LIN {X 55.448,Y -40.335,Z -83.216,A -90.000,B 90.000,C 0.000} C_DIS
LIN {X 55.688,Y -40.322,Z -83.552,A -90.000,B 90.000,C 0.000} C_DIS
LIN {X 55.796,Y -40.317,Z -83.715,A -90.000,B 90.000,C 0.000} C_DIS
LIN {X 55.903,Y -40.312,Z -83.888,A -90.000,B 90.000,C 0.000} C_DIS
LIN {X 55.980,Y -40.309,Z -84.022,A -90.000,B 90.000,C 0.000} C_DIS
LIN {X 56.380,Y -40.279,Z -84.724,A -90.000,B 90.000,C 0.000} C_DIS
LIN {X 56.567,Y -40.275,Z -85.049,A -90.000,B 90.000,C 0.000} C_DIS
LIN {X 56.659,Y -40.271,Z -85.172,A -90.000,B 90.000,C 0.000} C_DIS
LIN {X 56.815,Y -40.265,Z -85.391,A -90.000,B 90.000,C 0.000} C_DIS
LIN {X 56.970,Y -40.260,Z -85.627,A -90.000,B 90.000,C 0.000} C_DIS
LIN {X 57.075,Y -40.256,Z -85.792,A -90.000,B 90.000,C 0.000} C_DIS
LIN {X 58.077,Y -40.178,Z -87.383,A -90.000,B 90.000,C 0.000} C_DIS
LIN {X 58.154,Y -40.176,Z -87.509,A -90.000,B 90.000,C 0.000} C_DIS
LIN {X 58.234,Y -40.175,Z -87.644,A -90.000,B 90.000,C 0.000} C_DIS
LIN {X 58.357,Y -40.178,Z -87.857,A -90.000,B 90.000,C 0.000} C_DIS
LIN {X 58.489,Y -40.182,Z -88.102,A -90.000,B 90.000,C 0.000} C_DIS
LIN {X 58.598,Y -40.187,Z -88.331,A -90.000,B 90.000,C 0.000} C_DIS
LIN {X 58.752,Y -40.195,Z -88.665,A -90.000,B 90.000,C 0.000} C_DIS
LIN {X 58.752,Y -60.000,Z -88.665,A -90.000,B 90.000,C 0.000} C_DIS
LIN {X 62.631,Y -60.000,Z -64.637,A -90.000,B 90.000,C 0.000} C_DIS
LIN {X 62.631,Y -39.308,Z -64.637,A -90.000,B 90.000,C 0.000} C_DIS
LIN {X 62.803,Y -39.336,Z -65.056,A -90.000,B 90.000,C 0.000} C_DIS
LIN {X 62.966,Y -39.374,Z -65.497,A -90.000,B 90.000,C 0.000} C_DIS
LIN {X 63.006,Y -39.387,Z -65.615,A -90.000,B 90.000,C 0.000} C_DIS
LIN {X 63.056,Y -39.406,Z -65.776,A -90.000,B 90.000,C 0.000} C_DIS
LIN {X 63.115,Y -39.421,Z -65.986,A -90.000,B 90.000,C 0.000} C_DIS
LIN {X 63.170,Y -39.449,Z -66.179,A -90.000,B 90.000,C 0.000} C_DIS
LIN {X 63.215,Y -39.481,Z -66.369,A -90.000,B 90.000,C 0.000} C_DIS
LIN {X 63.277,Y -39.540,Z -66.686,A -90.000,B 90.000,C 0.000} C_DIS
LIN {X 63.366,Y -39.573,Z -66.956,A -90.000,B 90.000,C 0.000} C_DIS
LIN {X 63.448,Y -39.581,Z -67.122,A -90.000,B 90.000,C 0.000} C_DIS
LIN {X 63.626,Y -39.622,Z -67.462,A -90.000,B 90.000,C 0.000} C_DIS
LIN {X 63.736,Y -39.653,Z -67.698,A -90.000,B 90.000,C 0.000} C_DIS
LIN {X 63.814,Y -39.679,Z -67.903,A -90.000,B 90.000,C 0.000} C_DIS
LIN {X 63.888,Y -39.711,Z -68.118,A -90.000,B 90.000,C 0.000} C_DIS
LIN {X 63.960,Y -39.739,Z -68.344,A -90.000,B 90.000,C 0.000} C_DIS
LIN {X 64.010,Y -39.762,Z -68.538,A -90.000,B 90.000,C 0.000} C_DIS
LIN {X 64.032,Y -39.775,Z -68.642,A -90.000,B 90.000,C 0.000} C_DIS
LIN {X 64.060,Y -39.804,Z -68.761,A -90.000,B 90.000,C 0.000} C_DIS
LIN {X 64.106,Y -39.865,Z -68.997,A -90.000,B 90.000,C 0.000} C_DIS
LIN {X 64.202,Y -39.871,Z -69.126,A -90.000,B 90.000,C 0.000} C_DIS
LIN {X 64.331,Y -39.885,Z -69.319,A -90.000,B 90.000,C 0.000} C_DIS
LIN {X 64.452,Y -39.896,Z -69.517,A -90.000,B 90.000,C 0.000} C_DIS
LIN {X 64.575,Y -39.927,Z -69.720,A -90.000,B 90.000,C 0.000} C_DIS
LIN {X 64.644,Y -39.949,Z -69.846,A -90.000,B 90.000,C 0.000} C_DIS
LIN {X 64.711,Y -39.973,Z -69.977,A -90.000,B 90.000,C 0.000} C_DIS
LIN {X 64.741,Y -39.985,Z -70.038,A -90.000,B 90.000,C 0.000} C_DIS
LIN {X 64.793,Y -40.011,Z -70.157,A -90.000,B 90.000,C 0.000} C_DIS
LIN {X 64.862,Y -40.038,Z -70.334,A -90.000,B 90.000,C 0.000} C_DIS
LIN {X 64.948,Y -40.071,Z -70.569,A -90.000,B 90.000,C 0.000} C_DIS
LIN {X 65.029,Y -40.110,Z -70.831,A -90.000,B 90.000,C 0.000} C_DIS
LIN {X 65.095,Y -40.142,Z -71.055,A -90.000,B 90.000,C 0.000} C_DIS
LIN {X 65.138,Y -40.181,Z -71.197,A -90.000,B 90.000,C 0.000} C_DIS
LIN {X 65.489,Y -40.180,Z -71.479,A -90.000,B 90.000,C 0.000} C_DIS
LIN {X 65.574,Y -40.181,Z -71.552,A -90.000,B 90.000,C 0.000} C_DIS
LIN {X 65.793,Y -40.190,Z -71.768,A -90.000,B 90.000,C 0.000} C_DIS
LIN {X 65.900,Y -40.190,Z -71.880,A -90.000,B 90.000,C 0.000} C_DIS
LIN {X 65.920,Y -40.190,Z -71.903,A -90.000,B 90.000,C 0.000} C_DIS
LIN {X 66.214,Y -40.123,Z -72.021,A -90.000,B 90.000,C 0.000} C_DIS
LIN {X 66.578,Y -40.065,Z -72.162,A -90.000,B 90.000,C 0.000} C_DIS
LIN {X 66.676,Y -40.051,Z -72.204,A -90.000,B 90.000,C 0.000} C_DIS
LIN {X 66.897,Y -40.022,Z -72.304,A -90.000,B 90.000,C 0.000} C_DIS
LIN {X 67.010,Y -40.009,Z -72.360,A -90.000,B 90.000,C 0.000} C_DIS
LIN {X 67.972,Y -39.914,Z -72.867,A -90.000,B 90.000,C 0.000} C_DIS
LIN {X 68.175,Y -39.891,Z -72.982,A -90.000,B 90.000,C 0.000} C_DIS
LIN {X 68.701,Y -39.841,Z -73.302,A -90.000,B 90.000,C 0.000} C_DIS
LIN {X 68.861,Y -39.829,Z -73.407,A -90.000,B 90.000,C 0.000} C_DIS
LIN {X 68.964,Y -39.823,Z -73.479,A -90.000,B 90.000,C 0.000} C_DIS
LIN {X 69.180,Y -39.815,Z -73.639,A -90.000,B 90.000,C 0.000} C_DIS
LIN {X 69.326,Y -39.812,Z -73.753,A -90.000,B 90.000,C 0.000} C_DIS
LIN {X 69.405,Y -39.811,Z -73.818,A -90.000,B 90.000,C 0.000} C_DIS
LIN {X 69.492,Y -39.812,Z -73.891,A -90.000,B 90.000,C 0.000} C_DIS
LIN {X 69.916,Y -39.830,Z -74.281,A -90.000,B 90.000,C 0.000} C_DIS
LIN {X 70.119,Y -39.790,Z -74.354,A -90.000,B 90.000,C 0.000} C_DIS
LIN {X 70.283,Y -39.762,Z -74.421,A -90.000,B 90.000,C 0.000} C_DIS
LIN {X 70.508,Y -39.729,Z -74.526,A -90.000,B 90.000,C 0.000} C_DIS
LIN {X 70.711,Y -39.701,Z -74.624,A -90.000,B 90.000,C 0.000} C_DIS
LIN {X 71.011,Y -39.667,Z -74.789,A -90.000,B 90.000,C 0.000} C_DIS
LIN {X 71.174,Y -39.654,Z -74.889,A -90.000,B 90.000,C 0.000} C_DIS
LIN {X 71.373,Y -39.643,Z -75.025,A -90.000,B 90.000,C 0.000} C_DIS
LIN {X 71.608,Y -39.629,Z -75.193,A -90.000,B 90.000,C 0.000} C_DIS
LIN {X 71.729,Y -39.619,Z -75.284,A -90.000,B 90.000,C 0.000} C_DIS
LIN {X 72.076,Y -39.581,Z -75.549,A -90.000,B 90.000,C 0.000} C_DIS
LIN {X 72.224,Y -39.570,Z -75.678,A -90.000,B 90.000,C 0.000} C_DIS
LIN {X 72.416,Y -39.557,Z -75.848,A -90.000,B 90.000,C 0.000} C_DIS
LIN {X 72.547,Y -39.553,Z -75.976,A -90.000,B 90.000,C 0.000} C_DIS
LIN {X 72.645,Y -39.552,Z -76.075,A -90.000,B 90.000,C 0.000} C_DIS
LIN {X 72.773,Y -39.560,Z -76.196,A -90.000,B 90.000,C 0.000} C_DIS
LIN {X 72.854,Y -39.553,Z -76.248,A -90.000,B 90.000,C 0.000} C_DIS
LIN {X 73.182,Y -39.532,Z -76.475,A -90.000,B 90.000,C 0.000} C_DIS
LIN {X 73.340,Y -39.517,Z -76.596,A -90.000,B 90.000,C 0.000} C_DIS
LIN {X 73.415,Y -39.512,Z -76.659,A -90.000,B 90.000,C 0.000} C_DIS
LIN {X 73.579,Y -39.490,Z -76.774,A -90.000,B 90.000,C 0.000} C_DIS
LIN {X 73.871,Y -39.448,Z -76.998,A -90.000,B 90.000,C 0.000} C_DIS
LIN {X 74.097,Y -39.423,Z -77.189,A -90.000,B 90.000,C 0.000} C_DIS
LIN {X 74.181,Y -39.415,Z -77.265,A -90.000,B 90.000,C 0.000} C_DIS
LIN {X 74.301,Y -39.406,Z -77.378,A -90.000,B 90.000,C 0.000} C_DIS
LIN {X 74.531,Y -39.408,Z -77.577,A -90.000,B 90.000,C 0.000} C_DIS
LIN {X 74.759,Y -39.404,Z -77.780,A -90.000,B 90.000,C 0.000} C_DIS
LIN {X 74.822,Y -39.403,Z -77.835,A -90.000,B 90.000,C 0.000} C_DIS
LIN {X 75.001,Y -39.394,Z -77.985,A -90.000,B 90.000,C 0.000} C_DIS
LIN {X 75.071,Y -39.388,Z -78.045,A -90.000,B 90.000,C 0.000} C_DIS
LIN {X 75.136,Y -39.387,Z -78.100,A -90.000,B 90.000,C 0.000} C_DIS
LIN {X 75.196,Y -39.384,Z -78.154,A -90.000,B 90.000,C 0.000} C_DIS
LIN {X 75.547,Y -39.343,Z -78.421,A -90.000,B 90.000,C 0.000} C_DIS
LIN {X 75.912,Y -39.338,Z -78.674,A -90.000,B 90.000,C 0.000} C_DIS
LIN {X 76.049,Y -39.331,Z -78.780,A -90.000,B 90.000,C 0.000} C_DIS
LIN {X 76.147,Y -39.338,Z -78.854,A -90.000,B 90.000,C 0.000} C_DIS
LIN {X 76.292,Y -39.341,Z -78.955,A -90.000,B 90.000,C 0.000} C_DIS
LIN {X 76.399,Y -39.345,Z -79.035,A -90.000,B 90.000,C 0.000} C_DIS
LIN {X 76.474,Y -39.345,Z -79.072,A -90.000,B 90.000,C 0.000} C_DIS
LIN {X 76.612,Y -39.308,Z -79.080,A -90.000,B 90.000,C 0.000} C_DIS
LIN {X 76.612,Y -60.000,Z -79.080,A -90.000,B 90.000,C 0.000} C_DIS
LIN {X 88.646,Y -60.000,Z -102.744,A -90.000,B 90.000,C 0.000} C_DIS
LIN {X 88.646,Y -39.308,Z -102.744,A -90.000,B 90.000,C 0.000} C_DIS
LIN {X 88.487,Y -39.355,Z -102.950,A -90.000,B 90.000,C 0.000} C_DIS
LIN {X 88.363,Y -39.383,Z -103.144,A -90.000,B 90.000,C 0.000} C_DIS
LIN {X 88.211,Y -39.434,Z -103.399,A -90.000,B 90.000,C 0.000} C_DIS
LIN {X 88.135,Y -39.455,Z -103.567,A -90.000,B 90.000,C 0.000} C_DIS
LIN {X 88.144,Y -39.422,Z -103.771,A -90.000,B 90.000,C 0.000} C_DIS
LIN {X 88.186,Y -39.403,Z -104.002,A -90.000,B 90.000,C 0.000} C_DIS
LIN {X 88.227,Y -39.387,Z -104.294,A -90.000,B 90.000,C 0.000} C_DIS
LIN {X 88.233,Y -39.385,Z -104.347,A -90.000,B 90.000,C 0.000} C_DIS
LIN {X 88.314,Y -39.424,Z -105.037,A -90.000,B 90.000,C 0.000} C_DIS
LIN {X 88.419,Y -39.420,Z -105.520,A -90.000,B 90.000,C 0.000} C_DIS
LIN {X 88.449,Y -39.421,Z -105.676,A -90.000,B 90.000,C 0.000} C_DIS
LIN {X 88.476,Y -39.426,Z -105.847,A -90.000,B 90.000,C 0.000} C_DIS
LIN {X 88.504,Y -39.438,Z -106.079,A -90.000,B 90.000,C 0.000} C_DIS
LIN {X 88.535,Y -39.454,Z -106.359,A -90.000,B 90.000,C 0.000} C_DIS
LIN {X 88.548,Y -39.470,Z -106.548,A -90.000,B 90.000,C 0.000} C_DIS
LIN {X 88.551,Y -39.479,Z -106.637,A -90.000,B 90.000,C 0.000} C_DIS
LIN {X 88.548,Y -39.491,Z -106.855,A -90.000,B 90.000,C 0.000} C_DIS
LIN {X 88.543,Y -39.500,Z -106.987,A -90.000,B 90.000,C 0.000} C_DIS
LIN {X 88.531,Y -39.518,Z -107.213,A -90.000,B 90.000,C 0.000} C_DIS
LIN {X 88.570,Y -39.536,Z -108.068,A -90.000,B 90.000,C 0.000} C_DIS
LIN {X 88.572,Y -39.543,Z -108.276,A -90.000,B 90.000,C 0.000} C_DIS
LIN {X 88.570,Y -39.549,Z -108.401,A -90.000,B 90.000,C 0.000} C_DIS
LIN {X 88.562,Y -39.553,Z -108.539,A -90.000,B 90.000,C 0.000} C_DIS
LIN {X 88.541,Y -39.554,Z -108.748,A -90.000,B 90.000,C 0.000} C_DIS
LIN {X 88.482,Y -39.564,Z -109.136,A -90.000,B 90.000,C 0.000} C_DIS
LIN {X 88.466,Y -39.568,Z -109.229,A -90.000,B 90.000,C 0.000} C_DIS
LIN {X 88.427,Y -39.579,Z -109.423,A -90.000,B 90.000,C 0.000} C_DIS
LIN {X 88.395,Y -39.588,Z -109.560,A -90.000,B 90.000,C 0.000} C_DIS
LIN {X 88.352,Y -39.603,Z -109.716,A -90.000,B 90.000,C 0.000} C_DIS
LIN {X 88.195,Y -39.657,Z -110.247,A -90.000,B 90.000,C 0.000} C_DIS
LIN {X 88.083,Y -39.686,Z -110.755,A -90.000,B 90.000,C 0.000} C_DIS
LIN {X 88.036,Y -39.686,Z -110.940,A -90.000,B 90.000,C 0.000} C_DIS
LIN {X 87.935,Y -39.696,Z -111.368,A -90.000,B 90.000,C 0.000} C_DIS
LIN {X 87.898,Y -39.701,Z -111.506,A -90.000,B 90.000,C 0.000} C_DIS
LIN {X 87.857,Y -39.707,Z -111.652,A -90.000,B 90.000,C 0.000} C_DIS
LIN {X 87.827,Y -39.712,Z -111.749,A -90.000,B 90.000,C 0.000} C_DIS
LIN {X 87.739,Y -39.730,Z -112.014,A -90.000,B 90.000,C 0.000} C_DIS
LIN {X 87.648,Y -39.751,Z -112.263,A -90.000,B 90.000,C 0.000} C_DIS
LIN {X 87.392,Y -39.814,Z -112.904,A -90.000,B 90.000,C 0.000} C_DIS
LIN {X 87.199,Y -39.849,Z -113.373,A -90.000,B 90.000,C 0.000} C_DIS
LIN {X 86.963,Y -39.880,Z -114.044,A -90.000,B 90.000,C 0.000} C_DIS
LIN {X 86.838,Y -39.903,Z -114.404,A -90.000,B 90.000,C 0.000} C_DIS
LIN {X 86.484,Y -39.977,Z -115.313,A -90.000,B 90.000,C 0.000} C_DIS
LIN {X 86.191,Y -40.045,Z -116.068,A -90.000,B 90.000,C 0.000} C_DIS
LIN {X 86.080,Y -40.068,Z -116.381,A -90.000,B 90.000,C 0.000} C_DIS
LIN {X 85.781,Y -40.113,Z -117.455,A -90.000,B 90.000,C 0.000} C_DIS
LIN {X 85.664,Y -40.158,Z -117.908,A -90.000,B 90.000,C 0.000} C_DIS
LIN {X 85.654,Y -40.148,Z -119.002,A -90.000,B 90.000,C 0.000} C_DIS
LIN {X 85.738,Y -40.106,Z -119.512,A -90.000,B 90.000,C 0.000} C_DIS
LIN {X 85.882,Y -40.072,Z -120.318,A -90.000,B 90.000,C 0.000} C_DIS
LIN {X 85.916,Y -40.064,Z -120.518,A -90.000,B 90.000,C 0.000} C_DIS
LIN {X 86.185,Y -39.981,Z -121.579,A -90.000,B 90.000,C 0.000} C_DIS
LIN {X 86.320,Y -39.951,Z -122.101,A -90.000,B 90.000,C 0.000} C_DIS
LIN {X 86.350,Y -39.944,Z -122.221,A -90.000,B 90.000,C 0.000} C_DIS
LIN {X 86.375,Y -39.939,Z -122.333,A -90.000,B 90.000,C 0.000} C_DIS
LIN {X 86.420,Y -39.933,Z -122.564,A -90.000,B 90.000,C 0.000} C_DIS
LIN {X 86.439,Y -39.931,Z -122.680,A -90.000,B 90.000,C 0.000} C_DIS
LIN {X 86.466,Y -39.930,Z -122.867,A -90.000,B 90.000,C 0.000} C_DIS
LIN {X 86.538,Y -39.915,Z -123.170,A -90.000,B 90.000,C 0.000} C_DIS
LIN {X 86.605,Y -39.894,Z -123.462,A -90.000,B 90.000,C 0.000} C_DIS
LIN {X 86.698,Y -39.857,Z -123.886,A -90.000,B 90.000,C 0.000} C_DIS
LIN {X 86.776,Y -39.837,Z -124.221,A -90.000,B 90.000,C 0.000} C_DIS
LIN {X 86.837,Y -39.825,Z -124.544,A -90.000,B 90.000,C 0.000} C_DIS
LIN {X 86.851,Y -39.823,Z -124.642,A -90.000,B 90.000,C 0.000} C_DIS
LIN {X 86.911,Y -39.820,Z -125.137,A -90.000,B 90.000,C 0.000} C_DIS
LIN {X 86.942,Y -39.814,Z -125.415,A -90.000,B 90.000,C 0.000} C_DIS
LIN {X 87.002,Y -39.789,Z -125.978,A -90.000,B 90.000,C 0.000} C_DIS
LIN {X 87.037,Y -39.776,Z -126.427,A -90.000,B 90.000,C 0.000} C_DIS
LIN {X 87.043,Y -39.773,Z -126.548,A -90.000,B 90.000,C 0.000} C_DIS
LIN {X 87.059,Y -39.743,Z -127.669,A -90.000,B 90.000,C 0.000} C_DIS
LIN {X 87.070,Y -39.717,Z -128.497,A -90.000,B 90.000,C 0.000} C_DIS
LIN {X 87.067,Y -39.711,Z -128.686,A -90.000,B 90.000,C 0.000} C_DIS
LIN {X 87.033,Y -39.699,Z -129.362,A -90.000,B 90.000,C 0.000} C_DIS
LIN {X 87.016,Y -39.689,Z -129.846,A -90.000,B 90.000,C 0.000} C_DIS
LIN {X 86.985,Y -39.668,Z -130.819,A -90.000,B 90.000,C 0.000} C_DIS
LIN {X 86.968,Y -39.663,Z -131.089,A -90.000,B 90.000,C 0.000} C_DIS
LIN {X 86.930,Y -39.657,Z -131.584,A -90.000,B 90.000,C 0.000} C_DIS
LIN {X 86.917,Y -39.657,Z -131.766,A -90.000,B 90.000,C 0.000} C_DIS
LIN {X 86.865,Y -39.630,Z -133.147,A -90.000,B 90.000,C 0.000} C_DIS
LIN {X 86.850,Y -39.626,Z -133.400,A -90.000,B 90.000,C 0.000} C_DIS
LIN {X 86.798,Y -39.618,Z -134.106,A -90.000,B 90.000,C 0.000} C_DIS
LIN {X 86.786,Y -39.617,Z -134.285,A -90.000,B 90.000,C 0.000} C_DIS
LIN {X 86.751,Y -39.607,Z -135.000,A -90.000,B 90.000,C 0.000} C_DIS
LIN {X 86.727,Y -39.581,Z -136.202,A -90.000,B 90.000,C 0.000} C_DIS
LIN {X 86.713,Y -39.568,Z -136.863,A -90.000,B 90.000,C 0.000} C_DIS
LIN {X 86.705,Y -39.563,Z -137.178,A -90.000,B 90.000,C 0.000} C_DIS
LIN {X 86.656,Y -39.546,Z -138.299,A -90.000,B 90.000,C 0.000} C_DIS
LIN {X 86.648,Y -39.537,Z -138.633,A -90.000,B 90.000,C 0.000} C_DIS
LIN {X 86.609,Y -39.500,Z -140.528,A -90.000,B 90.000,C 0.000} C_DIS
LIN {X 86.528,Y -39.476,Z -142.113,A -90.000,B 90.000,C 0.000} C_DIS
LIN {X 86.512,Y -39.466,Z -142.548,A -90.000,B 90.000,C 0.000} C_DIS
LIN {X 86.459,Y -39.436,Z -144.152,A -90.000,B 90.000,C 0.000} C_DIS
LIN {X 86.446,Y -39.434,Z -144.366,A -90.000,B 90.000,C 0.000} C_DIS
LIN {X 86.309,Y -39.403,Z -146.328,A -90.000,B 90.000,C 0.000} C_DIS
LIN {X 86.274,Y -39.391,Z -146.931,A -90.000,B 90.000,C 0.000} C_DIS
LIN {X 86.210,Y -39.372,Z -148.070,A -90.000,B 90.000,C 0.000} C_DIS
LIN {X 86.178,Y -39.370,Z -148.420,A -90.000,B 90.000,C 0.000} C_DIS
LIN {X 86.058,Y -39.356,Z -149.672,A -90.000,B 90.000,C 0.000} C_DIS
LIN {X 85.954,Y -39.340,Z -150.710,A -90.000,B 90.000,C 0.000} C_DIS
LIN {X 85.844,Y -39.315,Z -151.917,A -90.000,B 90.000,C 0.000} C_DIS
LIN {X 85.811,Y -39.311,Z -152.221,A -90.000,B 90.000,C 0.000} C_DIS
LIN {X 85.781,Y -39.308,Z -152.460,A -90.000,B 90.000,C 0.000} C_DIS
LIN {X 85.781,Y -60.000,Z -152.460,A -90.000,B 90.000,C 0.000} C_DIS
LIN {X 87.625,Y -60.000,Z -117.678,A -90.000,B 90.000,C 0.000} C_DIS
LIN {X 87.625,Y -39.308,Z -117.678,A -90.000,B 90.000,C 0.000} C_DIS
LIN {X 87.494,Y -39.355,Z -118.185,A -90.000,B 90.000,C 0.000} C_DIS
LIN {X 87.487,Y -39.346,Z -118.824,A -90.000,B 90.000,C 0.000} C_DIS
LIN {X 87.560,Y -39.308,Z -119.270,A -90.000,B 90.000,C 0.000} C_DIS
LIN {X 87.560,Y -60.000,Z -119.270,A -90.000,B 90.000,C 0.000} C_DIS
LIN {X 30.587,Y -60.000,Z -77.495,A -90.000,B 90.000,C 0.000} C_DIS
LIN {X 30.587,Y -41.056,Z -77.495,A -90.000,B 90.000,C 0.000} C_DIS
LIN {X 30.404,Y -41.070,Z -77.561,A -90.000,B 90.000,C 0.000} C_DIS
LIN {X 30.295,Y -41.077,Z -77.600,A -90.000,B 90.000,C 0.000} C_DIS
LIN {X 29.998,Y -41.099,Z -77.706,A -90.000,B 90.000,C 0.000} C_DIS
LIN {X 29.486,Y -41.132,Z -77.891,A -90.000,B 90.000,C 0.000} C_DIS
LIN {X 29.537,Y -41.137,Z -77.762,A -90.000,B 90.000,C 0.000} C_DIS
LIN {X 29.558,Y -41.139,Z -77.701,A -90.000,B 90.000,C 0.000} C_DIS
LIN {X 29.594,Y -41.142,Z -77.571,A -90.000,B 90.000,C 0.000} C_DIS
LIN {X 29.625,Y -41.143,Z -77.418,A -90.000,B 90.000,C 0.000} C_DIS
LIN {X 29.640,Y -41.142,Z -77.302,A -90.000,B 90.000,C 0.000} C_DIS
LIN {X 29.650,Y -41.139,Z -77.160,A -90.000,B 90.000,C 0.000} C_DIS
LIN {X 29.651,Y -41.136,Z -77.100,A -90.000,B 90.000,C 0.000} C_DIS
LIN {X 29.649,Y -41.132,Z -77.002,A -90.000,B 90.000,C 0.000} C_DIS
LIN {X 29.639,Y -41.122,Z -76.875,A -90.000,B 90.000,C 0.000} C_DIS
LIN {X 29.626,Y -41.109,Z -76.782,A -90.000,B 90.000,C 0.000} C_DIS
LIN {X 29.598,Y -41.091,Z -76.645,A -90.000,B 90.000,C 0.000} C_DIS
LIN {X 29.529,Y -41.057,Z -76.375,A -90.000,B 90.000,C 0.000} C_DIS
LIN {X 29.515,Y -41.048,Z -76.323,A -90.000,B 90.000,C 0.000} C_DIS
LIN {X 29.477,Y -41.023,Z -76.201,A -90.000,B 90.000,C 0.000} C_DIS
LIN {X 29.425,Y -41.003,Z -76.063,A -90.000,B 90.000,C 0.000} C_DIS
LIN {X 29.393,Y -40.994,Z -75.990,A -90.000,B 90.000,C 0.000} C_DIS
LIN {X 29.532,Y -41.014,Z -76.194,A -90.000,B 90.000,C 0.000} C_DIS
LIN {X 29.643,Y -41.043,Z -76.364,A -90.000,B 90.000,C 0.000} C_DIS
LIN {X 29.810,Y -41.063,Z -76.611,A -90.000,B 90.000,C 0.000} C_DIS
LIN {X 30.025,Y -41.086,Z -76.913,A -90.000,B 90.000,C 0.000} C_DIS
LIN {X 30.053,Y -41.086,Z -76.949,A -90.000,B 90.000,C 0.000} C_DIS
LIN {X 30.138,Y -41.086,Z -77.050,A -90.000,B 90.000,C 0.000} C_DIS
LIN {X 30.340,Y -41.074,Z -77.258,A -90.000,B 90.000,C 0.000} C_DIS
LIN {X 30.433,Y -41.067,Z -77.354,A -90.000,B 90.000,C 0.000} C_DIS
LIN {X 30.499,Y -41.061,Z -77.417,A -90.000,B 90.000,C 0.000} C_DIS
LIN {X 30.587,Y -41.056,Z -77.495,A -90.000,B 90.000,C 0.000} C_DIS
LIN {X 30.587,Y -60.000,Z -77.495,A -90.000,B 90.000,C 0.000} C_DIS
LIN {X -30.129,Y -60.000,Z -90.405,A -90.000,B 90.000,C 0.000} C_DIS
LIN {X -30.129,Y -39.308,Z -90.405,A -90.000,B 90.000,C 0.000} C_DIS
LIN {X -30.060,Y -39.322,Z -90.255,A -90.000,B 90.000,C 0.000} C_DIS
LIN {X -30.026,Y -39.329,Z -90.188,A -90.000,B 90.000,C 0.000} C_DIS
LIN {X -29.675,Y -39.377,Z -89.547,A -90.000,B 90.000,C 0.000} C_DIS
LIN {X -29.319,Y -39.432,Z -88.890,A -90.000,B 90.000,C 0.000} C_DIS
LIN {X -29.145,Y -39.454,Z -88.576,A -90.000,B 90.000,C 0.000} C_DIS
LIN {X -28.986,Y -39.471,Z -88.271,A -90.000,B 90.000,C 0.000} C_DIS
LIN {X -28.868,Y -39.480,Z -88.057,A -90.000,B 90.000,C 0.000} C_DIS
LIN {X -28.612,Y -39.494,Z -87.640,A -90.000,B 90.000,C 0.000} C_DIS
LIN {X -28.327,Y -39.516,Z -87.218,A -90.000,B 90.000,C 0.000} C_DIS
LIN {X -27.589,Y -39.556,Z -86.145,A -90.000,B 90.000,C 0.000} C_DIS
LIN {X -27.389,Y -39.559,Z -85.861,A -90.000,B 90.000,C 0.000} C_DIS
LIN {X -27.210,Y -39.558,Z -85.619,A -90.000,B 90.000,C 0.000} C_DIS
LIN {X -27.072,Y -39.562,Z -85.433,A -90.000,B 90.000,C 0.000} C_DIS
LIN {X -26.958,Y -39.567,Z -85.288,A -90.000,B 90.000,C 0.000} C_DIS
LIN {X -26.797,Y -39.578,Z -85.093,A -90.000,B 90.000,C 0.000} C_DIS
LIN {X -25.931,Y -39.615,Z -84.059,A -90.000,B 90.000,C 0.000} C_DIS
LIN {X -25.793,Y -39.625,Z -83.892,A -90.000,B 90.000,C 0.000} C_DIS
LIN {X -25.587,Y -39.631,Z -83.657,A -90.000,B 90.000,C 0.000} C_DIS
LIN {X -25.130,Y -39.647,Z -83.139,A -90.000,B 90.000,C 0.000} C_DIS
LIN {X -24.889,Y -39.658,Z -82.874,A -90.000,B 90.000,C 0.000} C_DIS
LIN {X -23.786,Y -39.723,Z -81.715,A -90.000,B 90.000,C 0.000} C_DIS
LIN {X -23.601,Y -39.731,Z -81.527,A -90.000,B 90.000,C 0.000} C_DIS
LIN {X -22.538,Y -39.776,Z -80.520,A -90.000,B 90.000,C 0.000} C_DIS
LIN {X -22.410,Y -39.782,Z -80.403,A -90.000,B 90.000,C 0.000} C_DIS
LIN {X -21.978,Y -39.811,Z -80.028,A -90.000,B 90.000,C 0.000} C_DIS
LIN {X -21.823,Y -39.824,Z -79.901,A -90.000,B 90.000,C 0.000} C_DIS
LIN {X -21.508,Y -39.845,Z -79.657,A -90.000,B 90.000,C 0.000} C_DIS
LIN {X -21.087,Y -39.864,Z -79.336,A -90.000,B 90.000,C 0.000} C_DIS
LIN {X -20.813,Y -39.876,Z -79.144,A -90.000,B 90.000,C 0.000} C_DIS
LIN {X -20.037,Y -39.903,Z -78.615,A -90.000,B 90.000,C 0.000} C_DIS
LIN {X -19.819,Y -39.906,Z -78.471,A -90.000,B 90.000,C 0.000} C_DIS
LIN {X -19.686,Y -39.909,Z -78.388,A -90.000,B 90.000,C 0.000} C_DIS
LIN {X -18.777,Y -39.945,Z -77.863,A -90.000,B 90.000,C 0.000} C_DIS
LIN {X -18.662,Y -39.950,Z -77.800,A -90.000,B 90.000,C 0.000} C_DIS
LIN {X -18.375,Y -39.959,Z -77.650,A -90.000,B 90.000,C 0.000} C_DIS
LIN {X -17.935,Y -39.967,Z -77.446,A -90.000,B 90.000,C 0.000} C_DIS
LIN {X -17.734,Y -39.970,Z -77.354,A -90.000,B 90.000,C 0.000} C_DIS
LIN {X -17.278,Y -39.959,Z -77.155,A -90.000,B 90.000,C 0.000} C_DIS
LIN {X -17.056,Y -39.958,Z -77.069,A -90.000,B 90.000,C 0.000} C_DIS
LIN {X -16.621,Y -39.961,Z -76.915,A -90.000,B 90.000,C 0.000} C_DIS
LIN {X -16.143,Y -39.952,Z -76.752,A -90.000,B 90.000,C 0.000} C_DIS
LIN {X -15.801,Y -39.950,Z -76.647,A -90.000,B 90.000,C 0.000} C_DIS
LIN {X -15.391,Y -39.949,Z -76.525,A -90.000,B 90.000,C 0.000} C_DIS
LIN {X -14.632,Y -39.931,Z -76.306,A -90.000,B 90.000,C 0.000} C_DIS
LIN {X -14.379,Y -39.922,Z -76.244,A -90.000,B 90.000,C 0.000} C_DIS
LIN {X -14.275,Y -39.920,Z -76.221,A -90.000,B 90.000,C 0.000} C_DIS
LIN {X -13.551,Y -39.908,Z -76.081,A -90.000,B 90.000,C 0.000} C_DIS
LIN {X -12.950,Y -39.892,Z -75.968,A -90.000,B 90.000,C 0.000} C_DIS
LIN {X -12.788,Y -39.890,Z -75.943,A -90.000,B 90.000,C 0.000} C_DIS
LIN {X -12.426,Y -39.882,Z -75.904,A -90.000,B 90.000,C 0.000} C_DIS
LIN {X -12.084,Y -39.870,Z -75.874,A -90.000,B 90.000,C 0.000} C_DIS
LIN {X -11.917,Y -39.862,Z -75.860,A -90.000,B 90.000,C 0.000} C_DIS
LIN {X -11.431,Y -39.830,Z -75.824,A -90.000,B 90.000,C 0.000} C_DIS
LIN {X -11.236,Y -39.819,Z -75.814,A -90.000,B 90.000,C 0.000} C_DIS
LIN {X -10.430,Y -39.787,Z -75.797,A -90.000,B 90.000,C 0.000} C_DIS
LIN {X -9.953,Y -39.776,Z -75.803,A -90.000,B 90.000,C 0.000} C_DIS
LIN {X -8.395,Y -39.730,Z -75.831,A -90.000,B 90.000,C 0.000} C_DIS
LIN {X -8.291,Y -39.728,Z -75.835,A -90.000,B 90.000,C 0.000} C_DIS
LIN {X -7.791,Y -39.723,Z -75.867,A -90.000,B 90.000,C 0.000} C_DIS
LIN {X -6.721,Y -39.690,Z -75.945,A -90.000,B 90.000,C 0.000} C_DIS
LIN {X -5.934,Y -39.664,Z -76.004,A -90.000,B 90.000,C 0.000} C_DIS
LIN {X -5.156,Y -39.625,Z -76.074,A -90.000,B 90.000,C 0.000} C_DIS
LIN {X -5.105,Y -39.623,Z -76.080,A -90.000,B 90.000,C 0.000} C_DIS
LIN {X -4.883,Y -39.616,Z -76.109,A -90.000,B 90.000,C 0.000} C_DIS
LIN {X -4.446,Y -39.605,Z -76.169,A -90.000,B 90.000,C 0.000} C_DIS
LIN {X -3.413,Y -39.590,Z -76.324,A -90.000,B 90.000,C 0.000} C_DIS
LIN {X -2.938,Y -39.575,Z -76.399,A -90.000,B 90.000,C 0.000} C_DIS
LIN {X -1.406,Y -39.549,Z -76.683,A -90.000,B 90.000,C 0.000} C_DIS
LIN {X -0.800,Y -39.544,Z -76.800,A -90.000,B 90.000,C 0.000} C_DIS
LIN {X 1.141,Y -39.538,Z -77.195,A -90.000,B 90.000,C 0.000} C_DIS
LIN {X 1.724,Y -39.530,Z -77.317,A -90.000,B 90.000,C 0.000} C_DIS
LIN {X 4.226,Y -39.506,Z -77.870,A -90.000,B 90.000,C 0.000} C_DIS
LIN {X 4.732,Y -39.506,Z -77.980,A -90.000,B 90.000,C 0.000} C_DIS
LIN {X 5.634,Y -39.510,Z -78.189,A -90.000,B 90.000,C 0.000} C_DIS
LIN {X 7.423,Y -39.500,Z -78.615,A -90.000,B 90.000,C 0.000} C_DIS
LIN {X 8.961,Y -39.505,Z -78.996,A -90.000,B 90.000,C 0.000} C_DIS
LIN {X 9.315,Y -39.511,Z -79.081,A -90.000,B 90.000,C 0.000} C_DIS
LIN {X 9.694,Y -39.520,Z -79.171,A -90.000,B 90.000,C 0.000} C_DIS
LIN {X 10.706,Y -39.530,Z -79.420,A -90.000,B 90.000,C 0.000} C_DIS
LIN {X 11.555,Y -39.547,Z -79.647,A -90.000,B 90.000,C 0.000} C_DIS
LIN {X 11.681,Y -39.548,Z -79.676,A -90.000,B 90.000,C 0.000} C_DIS
LIN {X 12.289,Y -39.555,Z -79.818,A -90.000,B 90.000,C 0.000} C_DIS
LIN {X 13.473,Y -39.635,Z -80.066,A -90.000,B 90.000,C 0.000} C_DIS
LIN {X 14.312,Y -39.692,Z -80.269,A -90.000,B 90.000,C 0.000} C_DIS
LIN {X 14.404,Y -39.698,Z -80.291,A -90.000,B 90.000,C 0.000} C_DIS
LIN {X 14.505,Y -39.704,Z -80.310,A -90.000,B 90.000,C 0.000} C_DIS
LIN {X 15.313,Y -39.783,Z -80.450,A -90.000,B 90.000,C 0.000} C_DIS
LIN {X 16.728,Y -39.925,Z -80.711,A -90.000,B 90.000,C 0.000} C_DIS
LIN {X 16.974,Y -39.951,Z -80.757,A -90.000,B 90.000,C 0.000} C_DIS
LIN {X 17.313,Y -39.984,Z -80.798,A -90.000,B 90.000,C 0.000} C_DIS
LIN {X 17.686,Y -40.026,Z -80.839,A -90.000,B 90.000,C 0.000} C_DIS
LIN {X 18.252,Y -40.088,Z -80.889,A -90.000,B 90.000,C 0.000} C_DIS
LIN {X 19.206,Y -40.187,Z -80.968,A -90.000,B 90.000,C 0.000} C_DIS
LIN {X 19.435,Y -40.210,Z -80.983,A -90.000,B 90.000,C 0.000} C_DIS
LIN {X 20.104,Y -40.288,Z -80.976,A -90.000,B 90.000,C 0.000} C_DIS
LIN {X 20.547,Y -40.337,Z -80.971,A -90.000,B 90.000,C 0.000} C_DIS
LIN {X 20.786,Y -40.361,Z -80.951,A -90.000,B 90.000,C 0.000} C_DIS
LIN {X 21.160,Y -40.394,Z -80.908,A -90.000,B 90.000,C 0.000} C_DIS
LIN {X 21.542,Y -40.422,Z -80.836,A -90.000,B 90.000,C 0.000} C_DIS
LIN {X 21.735,Y -40.426,Z -80.736,A -90.000,B 90.000,C 0.000} C_DIS
LIN {X 21.816,Y -40.423,Z -80.670,A -90.000,B 90.000,C 0.000} C_DIS
LIN {X 22.233,Y -40.410,Z -80.331,A -90.000,B 90.000,C 0.000} C_DIS
LIN {X 21.604,Y -40.287,Z -79.959,A -90.000,B 90.000,C 0.000} C_DIS
LIN {X 21.322,Y -40.232,Z -79.789,A -90.000,B 90.000,C 0.000} C_DIS
LIN {X 21.185,Y -40.204,Z -79.700,A -90.000,B 90.000,C 0.000} C_DIS
LIN {X 21.094,Y -40.185,Z -79.637,A -90.000,B 90.000,C 0.000} C_DIS
LIN {X 20.932,Y -40.149,Z -79.515,A -90.000,B 90.000,C 0.000} C_DIS
LIN {X 20.734,Y -40.103,Z -79.351,A -90.000,B 90.000,C 0.000} C_DIS
LIN {X 20.605,Y -40.070,Z -79.234,A -90.000,B 90.000,C 0.000} C_DIS
LIN {X 20.559,Y -40.058,Z -79.191,A -90.000,B 90.000,C 0.000} C_DIS
LIN {X 20.446,Y -40.026,Z -79.075,A -90.000,B 90.000,C 0.000} C_DIS
LIN {X 20.326,Y -39.994,Z -78.943,A -90.000,B 90.000,C 0.000} C_DIS
LIN {X 20.264,Y -39.977,Z -78.871,A -90.000,B 90.000,C 0.000} C_DIS
LIN {X 20.155,Y -39.944,Z -78.736,A -90.000,B 90.000,C 0.000} C_DIS
LIN {X 20.115,Y -39.928,Z -78.683,A -90.000,B 90.000,C 0.000} C_DIS
LIN {X 20.049,Y -39.898,Z -78.583,A -90.000,B 90.000,C 0.000} C_DIS
LIN {X 19.932,Y -39.841,Z -78.389,A -90.000,B 90.000,C 0.000} C_DIS
LIN {X 19.875,Y -39.811,Z -78.286,A -90.000,B 90.000,C 0.000} C_DIS
LIN {X 19.773,Y -39.748,Z -78.073,A -90.000,B 90.000,C 0.000} C_DIS
LIN {X 19.692,Y -39.693,Z -77.888,A -90.000,B 90.000,C 0.000} C_DIS
LIN {X 19.604,Y -39.628,Z -77.672,A -90.000,B 90.000,C 0.000} C_DIS
LIN {X 19.592,Y -39.618,Z -77.639,A -90.000,B 90.000,C 0.000} C_DIS
LIN {X 19.463,Y -39.654,Z -77.448,A -90.000,B 90.000,C 0.000} C_DIS
LIN {X 19.393,Y -39.679,Z -77.329,A -90.000,B 90.000,C 0.000} C_DIS
LIN {X 19.239,Y -39.744,Z -77.052,A -90.000,B 90.000,C 0.000} C_DIS
LIN {X 19.139,Y -39.802,Z -76.844,A -90.000,B 90.000,C 0.000} C_DIS
LIN {X 19.077,Y -39.841,Z -76.706,A -90.000,B 90.000,C 0.000} C_DIS
LIN {X 19.044,Y -39.860,Z -76.626,A -90.000,B 90.000,C 0.000} C_DIS
LIN {X 18.972,Y -39.907,Z -76.438,A -90.000,B 90.000,C 0.000} C_DIS
LIN {X 18.911,Y -39.957,Z -76.253,A -90.000,B 90.000,C 0.000} C_DIS
LIN {X 18.879,Y -39.991,Z -76.138,A -90.000,B 90.000,C 0.000} C_DIS
LIN {X 18.849,Y -40.026,Z -76.021,A -90.000,B 90.000,C 0.000} C_DIS
LIN {X 18.833,Y -40.047,Z -75.953,A -90.000,B 90.000,C 0.000} C_DIS
LIN {X 18.806,Y -40.088,Z -75.812,A -90.000,B 90.000,C 0.000} C_DIS
LIN {X 18.764,Y -40.172,Z -75.548,A -90.000,B 90.000,C 0.000} C_DIS
LIN {X 18.743,Y -40.224,Z -75.384,A -90.000,B 90.000,C 0.000} C_DIS
LIN {X 18.730,Y -40.272,Z -75.239,A -90.000,B 90.000,C 0.000} C_DIS
LIN {X 18.725,Y -40.334,Z -75.039,A -90.000,B 90.000,C 0.000} C_DIS
LIN {X 18.728,Y -40.374,Z -74.895,A -90.000,B 90.000,C 0.000} C_DIS
LIN {X 18.743,Y -40.431,Z -74.699,A -90.000,B 90.000,C 0.000} C_DIS
LIN {X 18.772,Y -40.487,Z -74.492,A -90.000,B 90.000,C 0.000} C_DIS
LIN {X 18.782,Y -40.503,Z -74.433,A -90.000,B 90.000,C 0.000} C_DIS
LIN {X 18.799,Y -40.523,Z -74.342,A -90.000,B 90.000,C 0.000} C_DIS
LIN {X 18.838,Y -40.556,Z -74.160,A -90.000,B 90.000,C 0.000} C_DIS
LIN {X 18.865,Y -40.576,Z -74.053,A -90.000,B 90.000,C 0.000} C_DIS
LIN {X 18.910,Y -40.605,Z -73.899,A -90.000,B 90.000,C 0.000} C_DIS
LIN {X 18.970,Y -40.639,Z -73.710,A -90.000,B 90.000,C 0.000} C_DIS
LIN {X 19.008,Y -40.650,Z -73.612,A -90.000,B 90.000,C 0.000} C_DIS
LIN {X 19.058,Y -40.664,Z -73.493,A -90.000,B 90.000,C 0.000} C_DIS
LIN {X 19.128,Y -40.677,Z -73.344,A -90.000,B 90.000,C 0.000} C_DIS
LIN {X 19.191,Y -40.689,Z -73.222,A -90.000,B 90.000,C 0.000} C_DIS
LIN {X 19.216,Y -40.693,Z -73.176,A -90.000,B 90.000,C 0.000} C_DIS
LIN {X 19.317,Y -40.707,Z -73.005,A -90.000,B 90.000,C 0.000} C_DIS
LIN {X 19.412,Y -40.710,Z -72.864,A -90.000,B 90.000,C 0.000} C_DIS
LIN {X 19.448,Y -40.712,Z -72.812,A -90.000,B 90.000,C 0.000} C_DIS
LIN {X 19.550,Y -40.709,Z -72.673,A -90.000,B 90.000,C 0.000} C_DIS
LIN {X 19.598,Y -40.707,Z -72.612,A -90.000,B 90.000,C 0.000} C_DIS
LIN {X 19.720,Y -40.696,Z -72.470,A -90.000,B 90.000,C 0.000} C_DIS
LIN {X 19.760,Y -40.692,Z -72.426,A -90.000,B 90.000,C 0.000} C_DIS
LIN {X 19.895,Y -40.673,Z -72.289,A -90.000,B 90.000,C 0.000} C_DIS
LIN {X 20.082,Y -40.636,Z -72.108,A -90.000,B 90.000,C 0.000} C_DIS
LIN {X 20.228,Y -40.617,Z -71.979,A -90.000,B 90.000,C 0.000} C_DIS
LIN {X 20.326,Y -40.606,Z -71.898,A -90.000,B 90.000,C 0.000} C_DIS
LIN {X 20.416,Y -40.596,Z -71.829,A -90.000,B 90.000,C 0.000} C_DIS
LIN {X 20.555,Y -40.579,Z -71.731,A -90.000,B 90.000,C 0.000} C_DIS
LIN {X 20.589,Y -40.576,Z -71.708,A -90.000,B 90.000,C 0.000} C_DIS
LIN {X 20.606,Y -40.573,Z -71.696,A -90.000,B 90.000,C 0.000} C_DIS
LIN {X 20.707,Y -40.556,Z -71.634,A -90.000,B 90.000,C 0.000} C_DIS
LIN {X 20.799,Y -40.541,Z -71.582,A -90.000,B 90.000,C 0.000} C_DIS
LIN {X 21.102,Y -40.472,Z -71.427,A -90.000,B 90.000,C 0.000} C_DIS
LIN {X 21.342,Y -40.419,Z -71.321,A -90.000,B 90.000,C 0.000} C_DIS
LIN {X 21.420,Y -40.394,Z -71.293,A -90.000,B 90.000,C 0.000} C_DIS
LIN {X 21.710,Y -40.312,Z -71.205,A -90.000,B 90.000,C 0.000} C_DIS
LIN {X 21.854,Y -40.270,Z -71.172,A -90.000,B 90.000,C 0.000} C_DIS
LIN {X 21.977,Y -40.237,Z -71.150,A -90.000,B 90.000,C 0.000} C_DIS
LIN {X 22.107,Y -40.196,Z -71.130,A -90.000,B 90.000,C 0.000} C_DIS
LIN {X 22.276,Y -40.140,Z -71.110,A -90.000,B 90.000,C 0.000} C_DIS
LIN {X 22.471,Y -40.080,Z -71.093,A -90.000,B 90.000,C 0.000} C_DIS
LIN {X 22.658,Y -40.025,Z -71.085,A -90.000,B 90.000,C 0.000} C_DIS
LIN {X 22.835,Y -39.976,Z -71.087,A -90.000,B 90.000,C 0.000} C_DIS
LIN {X 22.998,Y -39.923,Z -71.077,A -90.000,B 90.000,C 0.000} C_DIS
LIN {X 23.051,Y -39.946,Z -71.053,A -90.000,B 90.000,C 0.000} C_DIS
LIN {X 23.191,Y -39.996,Z -71.005,A -90.000,B 90.000,C 0.000} C_DIS
LIN {X 23.337,Y -40.047,Z -70.961,A -90.000,B 90.000,C 0.000} C_DIS
LIN {X 23.490,Y -40.100,Z -70.924,A -90.000,B 90.000,C 0.000} C_DIS
LIN {X 23.582,Y -40.127,Z -70.911,A -90.000,B 90.000,C 0.000} C_DIS
LIN {X 23.792,Y -40.187,Z -70.886,A -90.000,B 90.000,C 0.000} C_DIS
LIN {X 23.911,Y -40.221,Z -70.877,A -90.000,B 90.000,C 0.000} C_DIS
LIN {X 24.159,Y -40.290,Z -70.874,A -90.000,B 90.000,C 0.000} C_DIS
LIN {X 24.274,Y -40.312,Z -70.877,A -90.000,B 90.000,C 0.000} C_DIS
LIN {X 24.389,Y -40.335,Z -70.886,A -90.000,B 90.000,C 0.000} C_DIS
LIN {X 24.587,Y -40.373,Z -70.909,A -90.000,B 90.000,C 0.000} C_DIS
LIN {X 24.709,Y -40.395,Z -70.929,A -90.000,B 90.000,C 0.000} C_DIS
LIN {X 24.934,Y -40.437,Z -70.978,A -90.000,B 90.000,C 0.000} C_DIS
LIN {X 25.130,Y -40.474,Z -71.029,A -90.000,B 90.000,C 0.000} C_DIS
LIN {X 25.567,Y -40.549,Z -71.153,A -90.000,B 90.000,C 0.000} C_DIS
LIN {X 25.925,Y -40.612,Z -71.273,A -90.000,B 90.000,C 0.000} C_DIS
LIN {X 25.956,Y -40.617,Z -71.284,A -90.000,B 90.000,C 0.000} C_DIS
LIN {X 25.980,Y -40.621,Z -71.293,A -90.000,B 90.000,C 0.000} C_DIS
LIN {X 26.506,Y -40.660,Z -71.487,A -90.000,B 90.000,C 0.000} C_DIS
LIN {X 26.522,Y -40.638,Z -71.289,A -90.000,B 90.000,C 0.000} C_DIS
LIN {X 26.532,Y -40.621,Z -71.187,A -90.000,B 90.000,C 0.000} C_DIS
LIN {X 26.549,Y -40.594,Z -71.044,A -90.000,B 90.000,C 0.000} C_DIS
LIN {X 26.568,Y -40.568,Z -70.913,A -90.000,B 90.000,C 0.000} C_DIS
LIN {X 26.606,Y -40.530,Z -70.723,A -90.000,B 90.000,C 0.000} C_DIS
LIN {X 26.668,Y -40.447,Z -70.449,A -90.000,B 90.000,C 0.000} C_DIS
LIN {X 26.694,Y -40.415,Z -70.348,A -90.000,B 90.000,C 0.000} C_DIS
LIN {X 26.743,Y -40.362,Z -70.181,A -90.000,B 90.000,C 0.000} C_DIS
LIN {X 26.752,Y -40.352,Z -70.154,A -90.000,B 90.000,C 0.000} C_DIS
LIN {X 26.801,Y -40.290,Z -70.011,A -90.000,B 90.000,C 0.000} C_DIS
LIN {X 26.871,Y -40.214,Z -69.841,A -90.000,B 90.000,C 0.000} C_DIS
LIN {X 26.919,Y -40.168,Z -69.738,A -90.000,B 90.000,C 0.000} C_DIS
LIN {X 26.950,Y -40.134,Z -69.674,A -90.000,B 90.000,C 0.000} C_DIS
LIN {X 26.993,Y -40.085,Z -69.590,A -90.000,B 90.000,C 0.000} C_DIS
LIN {X 27.058,Y -40.014,Z -69.472,A -90.000,B 90.000,C 0.000} C_DIS
LIN {X 27.061,Y -39.947,Z -69.343,A -90.000,B 90.000,C 0.000} C_DIS
LIN {X 27.052,Y -39.911,Z -69.271,A -90.000,B 90.000,C 0.000} C_DIS
LIN {X 27.039,Y -39.796,Z -69.085,A -90.000,B 90.000,C 0.000} C_DIS
LIN {X 27.038,Y -39.681,Z -68.905,A -90.000,B 90.000,C 0.000} C_DIS
LIN {X 27.047,Y -39.560,Z -68.717,A -90.000,B 90.000,C 0.000} C_DIS
LIN {X 27.053,Y -39.509,Z -68.652,A -90.000,B 90.000,C 0.000} C_DIS
LIN {X 27.079,Y -39.368,Z -68.482,A -90.000,B 90.000,C 0.000} C_DIS
LIN {X 27.072,Y -39.351,Z -68.307,A -90.000,B 90.000,C 0.000} C_DIS
LIN {X 27.069,Y -39.332,Z -68.164,A -90.000,B 90.000,C 0.000} C_DIS
LIN {X 27.068,Y -39.308,Z -68.042,A -90.000,B 90.000,C 0.000} C_DIS
LIN {X 27.064,Y -39.286,Z -67.914,A -90.000,B 90.000,C 0.000} C_DIS
LIN {X 27.055,Y -39.245,Z -67.733,A -90.000,B 90.000,C 0.000} C_DIS
LIN {X 27.043,Y -39.220,Z -67.619,A -90.000,B 90.000,C 0.000} C_DIS
LIN {X 27.028,Y -39.196,Z -67.510,A -90.000,B 90.000,C 0.000} C_DIS
LIN {X 27.010,Y -39.171,Z -67.406,A -90.000,B 90.000,C 0.000} C_DIS
LIN {X 26.988,Y -39.146,Z -67.307,A -90.000,B 90.000,C 0.000} C_DIS
LIN {X 26.962,Y -39.122,Z -67.213,A -90.000,B 90.000,C 0.000} C_DIS
LIN {X 26.934,Y -39.098,Z -67.124,A -90.000,B 90.000,C 0.000} C_DIS
LIN {X 26.902,Y -39.074,Z -67.039,A -90.000,B 90.000,C 0.000} C_DIS
LIN {X 26.868,Y -39.051,Z -66.960,A -90.000,B 90.000,C 0.000} C_DIS
LIN {X 26.830,Y -39.027,Z -66.884,A -90.000,B 90.000,C 0.000} C_DIS
LIN {X 26.789,Y -39.004,Z -66.814,A -90.000,B 90.000,C 0.000} C_DIS
LIN {X 26.746,Y -38.981,Z -66.747,A -90.000,B 90.000,C 0.000} C_DIS
LIN {X 26.700,Y -38.958,Z -66.686,A -90.000,B 90.000,C 0.000} C_DIS
LIN {X 26.651,Y -38.935,Z -66.628,A -90.000,B 90.000,C 0.000} C_DIS
LIN {X 26.599,Y -38.913,Z -66.575,A -90.000,B 90.000,C 0.000} C_DIS
LIN {X 26.545,Y -38.891,Z -66.525,A -90.000,B 90.000,C 0.000} C_DIS
LIN {X 26.488,Y -38.869,Z -66.480,A -90.000,B 90.000,C 0.000} C_DIS
LIN {X 26.429,Y -38.847,Z -66.439,A -90.000,B 90.000,C 0.000} C_DIS
LIN {X 26.368,Y -38.826,Z -66.402,A -90.000,B 90.000,C 0.000} C_DIS
LIN {X 26.304,Y -38.805,Z -66.369,A -90.000,B 90.000,C 0.000} C_DIS
LIN {X 26.238,Y -38.784,Z -66.339,A -90.000,B 90.000,C 0.000} C_DIS
LIN {X 26.135,Y -38.753,Z -66.302,A -90.000,B 90.000,C 0.000} C_DIS
LIN {X 25.991,Y -38.713,Z -66.265,A -90.000,B 90.000,C 0.000} C_DIS
LIN {X 25.839,Y -38.674,Z -66.241,A -90.000,B 90.000,C 0.000} C_DIS
LIN {X 25.681,Y -38.637,Z -66.231,A -90.000,B 90.000,C 0.000} C_DIS
LIN {X 25.599,Y -38.619,Z -66.230,A -90.000,B 90.000,C 0.000} C_DIS
LIN {X 25.431,Y -38.583,Z -66.238,A -90.000,B 90.000,C 0.000} C_DIS
LIN {X 25.258,Y -38.549,Z -66.258,A -90.000,B 90.000,C 0.000} C_DIS
LIN {X 25.079,Y -38.516,Z -66.289,A -90.000,B 90.000,C 0.000} C_DIS
LIN {X 24.897,Y -38.485,Z -66.331,A -90.000,B 90.000,C 0.000} C_DIS
LIN {X 24.711,Y -38.455,Z -66.382,A -90.000,B 90.000,C 0.000} C_DIS
LIN {X 24.615,Y -38.445,Z -66.407,A -90.000,B 90.000,C 0.000} C_DIS
LIN {X 24.517,Y -38.490,Z -66.430,A -90.000,B 90.000,C 0.000} C_DIS
LIN {X 24.421,Y -38.540,Z -66.464,A -90.000,B 90.000,C 0.000} C_DIS
LIN {X 24.228,Y -38.635,Z -66.538,A -90.000,B 90.000,C 0.000} C_DIS
LIN {X 24.130,Y -38.679,Z -66.577,A -90.000,B 90.000,C 0.000} C_DIS
LIN {X 23.935,Y -38.762,Z -66.663,A -90.000,B 90.000,C 0.000} C_DIS
LIN {X 23.640,Y -38.880,Z -66.803,A -90.000,B 90.000,C 0.000} C_DIS
LIN {X 23.444,Y -38.948,Z -66.904,A -90.000,B 90.000,C 0.000} C_DIS
LIN {X 23.248,Y -39.008,Z -67.011,A -90.000,B 90.000,C 0.000} C_DIS
LIN {X 23.054,Y -39.057,Z -67.122,A -90.000,B 90.000,C 0.000} C_DIS
LIN {X 22.957,Y -39.078,Z -67.180,A -90.000,B 90.000,C 0.000} C_DIS
LIN {X 22.766,Y -39.113,Z -67.297,A -90.000,B 90.000,C 0.000} C_DIS
LIN {X 22.577,Y -39.138,Z -67.418,A -90.000,B 90.000,C 0.000} C_DIS
LIN {X 22.484,Y -39.146,Z -67.480,A -90.000,B 90.000,C 0.000} C_DIS
LIN {X 22.300,Y -39.157,Z -67.605,A -90.000,B 90.000,C 0.000} C_DIS
LIN {X 22.121,Y -39.158,Z -67.731,A -90.000,B 90.000,C 0.000} C_DIS
LIN {X 21.946,Y -39.150,Z -67.859,A -90.000,B 90.000,C 0.000} C_DIS
LIN {X 21.777,Y -39.134,Z -67.988,A -90.000,B 90.000,C 0.000} C_DIS
LIN {X 21.613,Y -39.109,Z -68.116,A -90.000,B 90.000,C 0.000} C_DIS
LIN {X 21.457,Y -39.083,Z -68.244,A -90.000,B 90.000,C 0.000} C_DIS
LIN {X 21.307,Y -39.051,Z -68.371,A -90.000,B 90.000,C 0.000} C_DIS
LIN {X 21.165,Y -39.014,Z -68.496,A -90.000,B 90.000,C 0.000} C_DIS
LIN {X 21.031,Y -38.971,Z -68.619,A -90.000,B 90.000,C 0.000} C_DIS
LIN {X 20.906,Y -38.925,Z -68.738,A -90.000,B 90.000,C 0.000} C_DIS
LIN {X 20.876,Y -38.923,Z -68.768,A -90.000,B 90.000,C 0.000} C_DIS
LIN {X 20.736,Y -39.060,Z -68.911,A -90.000,B 90.000,C 0.000} C_DIS
LIN {X 20.636,Y -39.163,Z -69.021,A -90.000,B 90.000,C 0.000} C_DIS
LIN {X 20.506,Y -39.303,Z -69.176,A -90.000,B 90.000,C 0.000} C_DIS
LIN {X 20.434,Y -39.387,Z -69.272,A -90.000,B 90.000,C 0.000} C_DIS
LIN {X 20.349,Y -39.492,Z -69.402,A -90.000,B 90.000,C 0.000} C_DIS
LIN {X 20.311,Y -39.549,Z -69.479,A -90.000,B 90.000,C 0.000} C_DIS
LIN {X 20.286,Y -39.597,Z -69.548,A -90.000,B 90.000,C 0.000} C_DIS
LIN {X 20.276,Y -39.636,Z -69.608,A -90.000,B 90.000,C 0.000} C_DIS
LIN {X 20.278,Y -39.660,Z -69.648,A -90.000,B 90.000,C 0.000} C_DIS
LIN {X 20.285,Y -39.674,Z -69.671,A -90.000,B 90.000,C 0.000} C_DIS
LIN {X 20.302,Y -39.690,Z -69.701,A -90.000,B 90.000,C 0.000} C_DIS
LIN {X 20.318,Y -39.699,Z -69.718,A -90.000,B 90.000,C 0.000} C_DIS
LIN {X 20.350,Y -39.707,Z -69.739,A -90.000,B 90.000,C 0.000} C_DIS
LIN {X 20.377,Y -39.710,Z -69.750,A -90.000,B 90.000,C 0.000} C_DIS
LIN {X 20.425,Y -39.710,Z -69.760,A -90.000,B 90.000,C 0.000} C_DIS
LIN {X 20.461,Y -39.706,Z -69.763,A -90.000,B 90.000,C 0.000} C_DIS
LIN {X 20.547,Y -39.690,Z -69.760,A -90.000,B 90.000,C 0.000} C_DIS
LIN {X 20.651,Y -39.660,Z -69.745,A -90.000,B 90.000,C 0.000} C_DIS
LIN {X 20.773,Y -39.615,Z -69.716,A -90.000,B 90.000,C 0.000} C_DIS
LIN {X 20.842,Y -39.585,Z -69.696,A -90.000,B 90.000,C 0.000} C_DIS
LIN {X 20.916,Y -39.550,Z -69.673,A -90.000,B 90.000,C 0.000} C_DIS
LIN {X 21.080,Y -39.467,Z -69.615,A -90.000,B 90.000,C 0.000} C_DIS
LIN {X 21.365,Y -39.311,Z -69.500,A -90.000,B 90.000,C 0.000} C_DIS
LIN {X 21.476,Y -39.267,Z -69.466,A -90.000,B 90.000,C 0.000} C_DIS
LIN {X 21.587,Y -39.308,Z -69.415,A -90.000,B 90.000,C 0.000} C_DIS
LIN {X 21.742,Y -39.365,Z -69.344,A -90.000,B 90.000,C 0.000} C_DIS
LIN {X 21.877,Y -39.414,Z -69.289,A -90.000,B 90.000,C 0.000} C_DIS
LIN {X 22.052,Y -39.479,Z -69.230,A -90.000,B 90.000,C 0.000} C_DIS
LIN {X 22.159,Y -39.512,Z -69.201,A -90.000,B 90.000,C 0.000} C_DIS
LIN {X 22.289,Y -39.553,Z -69.172,A -90.000,B 90.000,C 0.000} C_DIS
LIN {X 22.373,Y -39.580,Z -69.155,A -90.000,B 90.000,C 0.000} C_DIS
LIN {X 22.498,Y -39.614,Z -69.135,A -90.000,B 90.000,C 0.000} C_DIS
LIN {X 22.613,Y -39.646,Z -69.122,A -90.000,B 90.000,C 0.000} C_DIS
LIN {X 22.770,Y -39.684,Z -69.074,A -90.000,B 90.000,C 0.000} C_DIS
LIN {X 22.938,Y -39.717,Z -69.029,A -90.000,B 90.000,C 0.000} C_DIS
LIN {X 23.108,Y -39.750,Z -68.993,A -90.000,B 90.000,C 0.000} C_DIS
LIN {X 23.243,Y -39.773,Z -68.967,A -90.000,B 90.000,C 0.000} C_DIS
LIN {X 23.439,Y -39.806,Z -68.942,A -90.000,B 90.000,C 0.000} C_DIS
LIN {X 23.583,Y -39.829,Z -68.928,A -90.000,B 90.000,C 0.000} C_DIS
LIN {X 23.747,Y -39.847,Z -68.915,A -90.000,B 90.000,C 0.000} C_DIS
LIN {X 23.971,Y -39.875,Z -68.908,A -90.000,B 90.000,C 0.000} C_DIS
LIN {X 24.288,Y -39.906,Z -68.915,A -90.000,B 90.000,C 0.000} C_DIS
LIN {X 24.413,Y -39.919,Z -68.921,A -90.000,B 90.000,C 0.000} C_DIS
LIN {X 24.552,Y -39.929,Z -68.933,A -90.000,B 90.000,C 0.000} C_DIS
LIN {X 24.788,Y -39.950,Z -68.962,A -90.000,B 90.000,C 0.000} C_DIS
LIN {X 24.956,Y -39.961,Z -68.987,A -90.000,B 90.000,C 0.000} C_DIS
LIN {X 25.049,Y -39.969,Z -69.004,A -90.000,B 90.000,C 0.000} C_DIS
LIN {X 25.051,Y -39.894,Z -68.824,A -90.000,B 90.000,C 0.000} C_DIS
LIN {X 25.057,Y -39.834,Z -68.678,A -90.000,B 90.000,C 0.000} C_DIS
LIN {X 25.070,Y -39.735,Z -68.471,A -90.000,B 90.000,C 0.000} C_DIS
LIN {X 25.092,Y -39.631,Z -68.279,A -90.000,B 90.000,C 0.000} C_DIS
LIN {X 25.081,Y -39.552,Z -68.131,A -90.000,B 90.000,C 0.000} C_DIS
LIN {X 25.076,Y -39.491,Z -68.015,A -90.000,B 90.000,C 0.000} C_DIS
LIN {X 25.075,Y -39.466,Z -67.973,A -90.000,B 90.000,C 0.000} C_DIS
LIN {X 25.080,Y -39.384,Z -67.837,A -90.000,B 90.000,C 0.000} C_DIS
LIN {X 25.093,Y -39.308,Z -67.726,A -90.000,B 90.000,C 0.000} C_DIS
LIN {X 25.093,Y -60.000,Z -67.726,A -90.000,B 90.000,C 0.000} C_DIS
LIN {X 16.997,Y -60.000,Z -74.977,A -90.000,B 90.000,C 0.000} C_DIS
LIN {X 16.997,Y -39.308,Z -74.977,A -90.000,B 90.000,C 0.000} C_DIS
LIN {X 16.989,Y -39.352,Z -74.866,A -90.000,B 90.000,C 0.000} C_DIS
LIN {X 16.986,Y -39.416,Z -74.666,A -90.000,B 90.000,C 0.000} C_DIS
LIN {X 16.988,Y -39.471,Z -74.499,A -90.000,B 90.000,C 0.000} C_DIS
LIN {X 17.004,Y -39.568,Z -74.218,A -90.000,B 90.000,C 0.000} C_DIS
LIN {X 17.011,Y -39.596,Z -74.142,A -90.000,B 90.000,C 0.000} C_DIS
LIN {X 17.050,Y -39.706,Z -73.815,A -90.000,B 90.000,C 0.000} C_DIS
LIN {X 17.088,Y -39.786,Z -73.574,A -90.000,B 90.000,C 0.000} C_DIS
LIN {X 17.119,Y -39.842,Z -73.409,A -90.000,B 90.000,C 0.000} C_DIS
LIN {X 17.155,Y -39.887,Z -73.261,A -90.000,B 90.000,C 0.000} C_DIS
LIN {X 17.241,Y -39.966,Z -72.962,A -90.000,B 90.000,C 0.000} C_DIS
LIN {X 17.257,Y -39.980,Z -72.914,A -90.000,B 90.000,C 0.000} C_DIS
LIN {X 17.336,Y -40.030,Z -72.697,A -90.000,B 90.000,C 0.000} C_DIS
LIN {X 17.386,Y -40.061,Z -72.573,A -90.000,B 90.000,C 0.000} C_DIS
LIN {X 17.465,Y -40.088,Z -72.401,A -90.000,B 90.000,C 0.000} C_DIS
LIN {X 17.531,Y -40.109,Z -72.268,A -90.000,B 90.000,C 0.000} C_DIS
LIN {X 17.595,Y -40.123,Z -72.151,A -90.000,B 90.000,C 0.000} C_DIS
LIN {X 17.675,Y -40.141,Z -72.014,A -90.000,B 90.000,C 0.000} C_DIS
LIN {X 17.734,Y -40.148,Z -71.917,A -90.000,B 90.000,C 0.000} C_DIS
LIN {X 17.882,Y -40.168,Z -71.693,A -90.000,B 90.000,C 0.000} C_DIS
LIN {X 18.042,Y -40.174,Z -71.473,A -90.000,B 90.000,C 0.000} C_DIS
LIN {X 18.169,Y -40.169,Z -71.318,A -90.000,B 90.000,C 0.000} C_DIS
LIN {X 18.224,Y -40.168,Z -71.252,A -90.000,B 90.000,C 0.000} C_DIS
LIN {X 18.353,Y -40.154,Z -71.110,A -90.000,B 90.000,C 0.000} C_DIS
LIN {X 18.415,Y -40.149,Z -71.046,A -90.000,B 90.000,C 0.000} C_DIS
LIN {X 18.609,Y -40.117,Z -70.854,A -90.000,B 90.000,C 0.000} C_DIS
LIN {X 18.756,Y -40.082,Z -70.718,A -90.000,B 90.000,C 0.000} C_DIS
LIN {X 18.963,Y -40.047,Z -70.539,A -90.000,B 90.000,C 0.000} C_DIS
LIN {X 19.149,Y -40.017,Z -70.392,A -90.000,B 90.000,C 0.000} C_DIS
LIN {X 19.204,Y -40.008,Z -70.351,A -90.000,B 90.000,C 0.000} C_DIS
LIN {X 19.268,Y -39.997,Z -70.305,A -90.000,B 90.000,C 0.000} C_DIS
LIN {X 19.485,Y -39.957,Z -70.159,A -90.000,B 90.000,C 0.000} C_DIS
LIN {X 19.712,Y -39.902,Z -70.028,A -90.000,B 90.000,C 0.000} C_DIS
LIN {X 19.843,Y -39.862,Z -69.962,A -90.000,B 90.000,C 0.000} C_DIS
LIN {X 20.193,Y -39.757,Z -69.795,A -90.000,B 90.000,C 0.000} C_DIS
LIN {X 20.430,Y -39.670,Z -69.706,A -90.000,B 90.000,C 0.000} C_DIS
LIN {X 20.550,Y -39.621,Z -69.666,A -90.000,B 90.000,C 0.000} C_DIS
LIN {X 20.679,Y -39.569,Z -69.628,A -90.000,B 90.000,C 0.000} C_DIS
LIN {X 20.917,Y -39.478,Z -69.568,A -90.000,B 90.000,C 0.000} C_DIS
LIN {X 21.070,Y -39.415,Z -69.536,A -90.000,B 90.000,C 0.000} C_DIS
LIN {X 21.230,Y -39.353,Z -69.508,A -90.000,B 90.000,C 0.000} C_DIS
LIN {X 21.351,Y -39.308,Z -69.491,A -90.000,B 90.000,C 0.000} C_DIS
LIN {X 21.470,Y -39.267,Z -69.476,A -90.000,B 90.000,C 0.000} C_DIS
LIN {X 21.686,Y -39.358,Z -69.453,A -90.000,B 90.000,C 0.000} C_DIS
LIN {X 21.878,Y -39.436,Z -69.442,A -90.000,B 90.000,C 0.000} C_DIS
LIN {X 22.044,Y -39.502,Z -69.441,A -90.000,B 90.000,C 0.000} C_DIS
LIN {X 22.118,Y -39.531,Z -69.444,A -90.000,B 90.000,C 0.000} C_DIS
LIN {X 22.249,Y -39.581,Z -69.458,A -90.000,B 90.000,C 0.000} C_DIS
LIN {X 22.357,Y -39.624,Z -69.482,A -90.000,B 90.000,C 0.000} C_DIS
LIN {X 22.424,Y -39.651,Z -69.505,A -90.000,B 90.000,C 0.000} C_DIS
LIN {X 22.479,Y -39.674,Z -69.534,A -90.000,B 90.000,C 0.000} C_DIS
LIN {X 22.508,Y -39.688,Z -69.555,A -90.000,B 90.000,C 0.000} C_DIS
LIN {X 22.544,Y -39.705,Z -69.591,A -90.000,B 90.000,C 0.000} C_DIS
LIN {X 22.568,Y -39.719,Z -69.631,A -90.000,B 90.000,C 0.000} C_DIS
LIN {X 22.581,Y -39.730,Z -69.675,A -90.000,B 90.000,C 0.000} C_DIS
LIN {X 22.583,Y -39.737,Z -69.723,A -90.000,B 90.000,C 0.000} C_DIS
LIN {X 22.579,Y -39.739,Z -69.758,A -90.000,B 90.000,C 0.000} C_DIS
LIN {X 22.571,Y -39.740,Z -69.793,A -90.000,B 90.000,C 0.000} C_DIS
LIN {X 22.541,Y -39.737,Z -69.870,A -90.000,B 90.000,C 0.000} C_DIS
LIN {X 22.495,Y -39.726,Z -69.951,A -90.000,B 90.000,C 0.000} C_DIS
LIN {X 22.432,Y -39.707,Z -70.038,A -90.000,B 90.000,C 0.000} C_DIS
LIN {X 22.355,Y -39.682,Z -70.130,A -90.000,B 90.000,C 0.000} C_DIS
LIN {X 22.263,Y -39.649,Z -70.227,A -90.000,B 90.000,C 0.000} C_DIS
LIN {X 22.213,Y -39.630,Z -70.276,A -90.000,B 90.000,C 0.000} C_DIS
LIN {X 22.158,Y -39.660,Z -70.327,A -90.000,B 90.000,C 0.000} C_DIS
LIN {X 22.040,Y -39.763,Z -70.430,A -90.000,B 90.000,C 0.000} C_DIS
LIN {X 21.911,Y -39.870,Z -70.537,A -90.000,B 90.000,C 0.000} C_DIS
LIN {X 21.769,Y -39.979,Z -70.646,A -90.000,B 90.000,C 0.000} C_DIS
LIN {X 21.695,Y -40.031,Z -70.701,A -90.000,B 90.000,C 0.000} C_DIS
LIN {X 21.539,Y -40.128,Z -70.813,A -90.000,B 90.000,C 0.000} C_DIS
LIN {X 21.457,Y -40.174,Z -70.869,A -90.000,B 90.000,C 0.000} C_DIS
LIN {X 21.287,Y -40.257,Z -70.983,A -90.000,B 90.000,C 0.000} C_DIS
LIN {X 21.109,Y -40.330,Z -71.097,A -90.000,B 90.000,C 0.000} C_DIS
LIN {X 20.923,Y -40.392,Z -71.212,A -90.000,B 90.000,C 0.000} C_DIS
LIN {X 20.731,Y -40.443,Z -71.326,A -90.000,B 90.000,C 0.000} C_DIS
LIN {X 20.533,Y -40.482,Z -71.439,A -90.000,B 90.000,C 0.000} C_DIS
LIN {X 20.330,Y -40.510,Z -71.552,A -90.000,B 90.000,C 0.000} C_DIS
LIN {X 20.123,Y -40.525,Z -71.662,A -90.000,B 90.000,C 0.000} C_DIS
LIN {X 19.912,Y -40.531,Z -71.771,A -90.000,B 90.000,C 0.000} C_DIS
LIN {X 19.698,Y -40.546,Z -71.877,A -90.000,B 90.000,C 0.000} C_DIS
LIN {X 19.483,Y -40.552,Z -71.980,A -90.000,B 90.000,C 0.000} C_DIS
LIN {X 19.266,Y -40.547,Z -72.080,A -90.000,B 90.000,C 0.000} C_DIS
LIN {X 19.049,Y -40.530,Z -72.176,A -90.000,B 90.000,C 0.000} C_DIS
LIN {X 18.833,Y -40.503,Z -72.267,A -90.000,B 90.000,C 0.000} C_DIS
LIN {X 18.725,Y -40.486,Z -72.311,A -90.000,B 90.000,C 0.000} C_DIS
LIN {X 18.617,Y -40.466,Z -72.353,A -90.000,B 90.000,C 0.000} C_DIS
LIN {X 18.404,Y -40.419,Z -72.434,A -90.000,B 90.000,C 0.000} C_DIS
LIN {X 18.193,Y -40.363,Z -72.510,A -90.000,B 90.000,C 0.000} C_DIS
LIN {X 17.985,Y -40.300,Z -72.579,A -90.000,B 90.000,C 0.000} C_DIS
LIN {X 17.782,Y -40.229,Z -72.641,A -90.000,B 90.000,C 0.000} C_DIS
LIN {X 17.682,Y -40.191,Z -72.670,A -90.000,B 90.000,C 0.000} C_DIS
LIN {X 17.487,Y -40.107,Z -72.722,A -90.000,B 90.000,C 0.000} C_DIS
LIN {X 17.298,Y -40.015,Z -72.765,A -90.000,B 90.000,C 0.000} C_DIS
LIN {X 17.206,Y -39.967,Z -72.784,A -90.000,B 90.000,C 0.000} C_DIS
LIN {X 17.027,Y -39.866,Z -72.815,A -90.000,B 90.000,C 0.000} C_DIS
LIN {X 16.856,Y -39.759,Z -72.837,A -90.000,B 90.000,C 0.000} C_DIS
LIN {X 16.695,Y -39.653,Z -72.850,A -90.000,B 90.000,C 0.000} C_DIS
LIN {X 16.543,Y -39.549,Z -72.853,A -90.000,B 90.000,C 0.000} C_DIS
LIN {X 16.401,Y -39.450,Z -72.846,A -90.000,B 90.000,C 0.000} C_DIS
LIN {X 16.271,Y -39.357,Z -72.827,A -90.000,B 90.000,C 0.000} C_DIS
LIN {X 16.210,Y -39.313,Z -72.814,A -90.000,B 90.000,C 0.000} C_DIS
LIN {X 16.152,Y -39.273,Z -72.798,A -90.000,B 90.000,C 0.000} C_DIS
LIN {X 16.097,Y -39.239,Z -72.779,A -90.000,B 90.000,C 0.000} C_DIS
LIN {X 16.046,Y -39.210,Z -72.756,A -90.000,B 90.000,C 0.000} C_DIS
LIN {X 15.998,Y -39.184,Z -72.731,A -90.000,B 90.000,C 0.000} C_DIS
LIN {X 15.954,Y -39.160,Z -72.703,A -90.000,B 90.000,C 0.000} C_DIS
LIN {X 15.894,Y -39.128,Z -72.655,A -90.000,B 90.000,C 0.000} C_DIS
LIN {X 15.859,Y -39.110,Z -72.618,A -90.000,B 90.000,C 0.000} C_DIS
LIN {X 15.827,Y -39.095,Z -72.579,A -90.000,B 90.000,C 0.000} C_DIS
LIN {X 15.787,Y -39.077,Z -72.513,A -90.000,B 90.000,C 0.000} C_DIS
LIN {X 15.756,Y -39.066,Z -72.440,A -90.000,B 90.000,C 0.000} C_DIS
LIN {X 15.735,Y -39.061,Z -72.358,A -90.000,B 90.000,C 0.000} C_DIS
LIN {X 15.726,Y -39.061,Z -72.299,A -90.000,B 90.000,C 0.000} C_DIS
LIN {X 15.721,Y -39.064,Z -72.237,A -90.000,B 90.000,C 0.000} C_DIS
LIN {X 15.723,Y -39.075,Z -72.136,A -90.000,B 90.000,C 0.000} C_DIS
LIN {X 15.730,Y -39.086,Z -72.064,A -90.000,B 90.000,C 0.000} C_DIS
LIN {X 15.742,Y -39.101,Z -71.988,A -90.000,B 90.000,C 0.000} C_DIS
LIN {X 15.769,Y -39.129,Z -71.867,A -90.000,B 90.000,C 0.000} C_DIS
LIN {X 15.822,Y -39.179,Z -71.692,A -90.000,B 90.000,C 0.000} C_DIS
LIN {X 15.897,Y -39.233,Z -71.500,A -90.000,B 90.000,C 0.000} C_DIS
LIN {X 15.993,Y -39.290,Z -71.291,A -90.000,B 90.000,C 0.000} C_DIS
LIN {X 16.049,Y -39.308,Z -71.179,A -90.000,B 90.000,C 0.000} C_DIS
LIN {X 16.138,Y -39.348,Z -71.008,A -90.000,B 90.000,C 0.000} C_DIS
LIN {X 16.228,Y -39.376,Z -70.851,A -90.000,B 90.000,C 0.000} C_DIS
LIN {X 16.321,Y -39.404,Z -70.700,A -90.000,B 90.000,C 0.000} C_DIS
LIN {X 16.392,Y -39.418,Z -70.591,A -90.000,B 90.000,C 0.000} C_DIS
LIN {X 16.525,Y -39.441,Z -70.395,A -90.000,B 90.000,C 0.000} C_DIS
LIN {X 16.583,Y -39.445,Z -70.316,A -90.000,B 90.000,C 0.000} C_DIS
LIN {X 16.712,Y -39.456,Z -70.149,A -90.000,B 90.000,C 0.000} C_DIS
LIN {X 16.861,Y -39.454,Z -69.972,A -90.000,B 90.000,C 0.000} C_DIS
LIN {X 16.934,Y -39.452,Z -69.888,A -90.000,B 90.000,C 0.000} C_DIS
LIN {X 17.143,Y -39.436,Z -69.669,A -90.000,B 90.000,C 0.000} C_DIS
LIN {X 17.378,Y -39.399,Z -69.439,A -90.000,B 90.000,C 0.000} C_DIS
LIN {X 17.457,Y -39.381,Z -69.368,A -90.000,B 90.000,C 0.000} C_DIS
LIN {X 17.611,Y -39.351,Z -69.238,A -90.000,B 90.000,C 0.000} C_DIS
LIN {X 17.683,Y -39.330,Z -69.179,A -90.000,B 90.000,C 0.000} C_DIS
LIN {X 17.789,Y -39.308,Z -69.096,A -90.000,B 90.000,C 0.000} C_DIS
LIN {X 17.789,Y -60.000,Z -69.096,A -90.000,B 90.000,C 0.000} C_DIS
LIN {X 13.365,Y -60.000,Z -78.022,A -90.000,B 90.000,C 0.000} C_DIS
LIN {X 13.365,Y -39.308,Z -78.022,A -90.000,B 90.000,C 0.000} C_DIS
LIN {X 13.957,Y -39.387,Z -78.141,A -90.000,B 90.000,C 0.000} C_DIS
LIN {X 14.759,Y -39.495,Z -78.330,A -90.000,B 90.000,C 0.000} C_DIS
LIN {X 14.821,Y -39.503,Z -78.345,A -90.000,B 90.000,C 0.000} C_DIS
LIN {X 15.188,Y -39.545,Z -78.408,A -90.000,B 90.000,C 0.000} C_DIS
LIN {X 15.770,Y -39.609,Z -78.509,A -90.000,B 90.000,C 0.000} C_DIS
LIN {X 17.125,Y -39.745,Z -78.760,A -90.000,B 90.000,C 0.000} C_DIS
LIN {X 17.293,Y -39.760,Z -78.791,A -90.000,B 90.000,C 0.000} C_DIS
LIN {X 17.907,Y -39.813,Z -78.862,A -90.000,B 90.000,C 0.000} C_DIS
LIN {X 17.938,Y -39.816,Z -78.865,A -90.000,B 90.000,C 0.000} C_DIS
LIN {X 17.834,Y -39.777,Z -78.623,A -90.000,B 90.000,C 0.000} C_DIS
LIN {X 17.814,Y -39.769,Z -78.573,A -90.000,B 90.000,C 0.000} C_DIS
LIN {X 17.752,Y -39.752,Z -78.478,A -90.000,B 90.000,C 0.000} C_DIS
LIN {X 17.650,Y -39.723,Z -78.310,A -90.000,B 90.000,C 0.000} C_DIS
LIN {X 17.485,Y -39.673,Z -78.011,A -90.000,B 90.000,C 0.000} C_DIS
LIN {X 17.464,Y -39.667,Z -77.972,A -90.000,B 90.000,C 0.000} C_DIS
LIN {X 17.407,Y -39.642,Z -77.850,A -90.000,B 90.000,C 0.000} C_DIS
LIN {X 17.304,Y -39.595,Z -77.612,A -90.000,B 90.000,C 0.000} C_DIS
LIN {X 17.225,Y -39.553,Z -77.405,A -90.000,B 90.000,C 0.000} C_DIS
LIN {X 17.173,Y -39.522,Z -77.248,A -90.000,B 90.000,C 0.000} C_DIS
LIN {X 17.145,Y -39.499,Z -77.149,A -90.000,B 90.000,C 0.000} C_DIS
LIN {X 17.119,Y -39.475,Z -77.054,A -90.000,B 90.000,C 0.000} C_DIS
LIN {X 17.090,Y -39.439,Z -76.924,A -90.000,B 90.000,C 0.000} C_DIS
LIN {X 17.051,Y -39.380,Z -76.707,A -90.000,B 90.000,C 0.000} C_DIS
LIN {X 17.037,Y -39.348,Z -76.594,A -90.000,B 90.000,C 0.000} C_DIS
LIN {X 17.026,Y -39.308,Z -76.455,A -90.000,B 90.000,C 0.000} C_DIS
LIN {X 17.026,Y -60.000,Z -76.455,A -90.000,B 90.000,C 0.000} C_DIS
LIN {X -26.369,Y -60.000,Z -134.517,A -90.000,B 90.000,C 0.000} C_DIS
LIN {X -26.369,Y -39.308,Z -134.517,A -90.000,B 90.000,C 0.000} C_DIS
LIN {X -26.416,Y -39.321,Z -134.425,A -90.000,B 90.000,C 0.000} C_DIS
LIN {X -26.693,Y -39.410,Z -133.851,A -90.000,B 90.000,C 0.000} C_DIS
LIN {X -27.060,Y -39.500,Z -133.040,A -90.000,B 90.000,C 0.000} C_DIS
LIN {X -27.151,Y -39.517,Z -132.816,A -90.000,B 90.000,C 0.000} C_DIS
LIN {X -27.588,Y -39.593,Z -131.700,A -90.000,B 90.000,C 0.000} C_DIS
LIN {X -27.836,Y -39.632,Z -131.076,A -90.000,B 90.000,C 0.000} C_DIS
LIN {X -28.397,Y -39.676,Z -129.828,A -90.000,B 90.000,C 0.000} C_DIS
LIN {X -28.479,Y -39.686,Z -129.631,A -90.000,B 90.000,C 0.000} C_DIS
LIN {X -28.563,Y -39.703,Z -129.407,A -90.000,B 90.000,C 0.000} C_DIS
LIN {X -28.641,Y -39.720,Z -129.184,A -90.000,B 90.000,C 0.000} C_DIS
LIN {X -28.929,Y -39.802,Z -128.285,A -90.000,B 90.000,C 0.000} C_DIS
LIN {X -28.943,Y -39.807,Z -128.239,A -90.000,B 90.000,C 0.000} C_DIS
LIN {X -29.050,Y -39.827,Z -127.910,A -90.000,B 90.000,C 0.000} C_DIS
LIN {X -29.282,Y -39.875,Z -127.173,A -90.000,B 90.000,C 0.000} C_DIS
LIN {X -29.381,Y -39.888,Z -126.842,A -90.000,B 90.000,C 0.000} C_DIS
LIN {X -29.509,Y -39.881,Z -126.529,A -90.000,B 90.000,C 0.000} C_DIS
LIN {X -29.590,Y -39.883,Z -126.339,A -90.000,B 90.000,C 0.000} C_DIS
LIN {X -29.694,Y -39.881,Z -126.089,A -90.000,B 90.000,C 0.000} C_DIS
LIN {X -29.964,Y -39.861,Z -125.425,A -90.000,B 90.000,C 0.000} C_DIS
LIN {X -30.113,Y -39.849,Z -125.063,A -90.000,B 90.000,C 0.000} C_DIS
LIN {X -30.197,Y -39.845,Z -124.837,A -90.000,B 90.000,C 0.000} C_DIS
LIN {X -30.278,Y -39.845,Z -124.595,A -90.000,B 90.000,C 0.000} C_DIS
LIN {X -30.527,Y -39.883,Z -123.876,A -90.000,B 90.000,C 0.000} C_DIS
LIN {X -30.595,Y -39.894,Z -123.678,A -90.000,B 90.000,C 0.000} C_DIS
LIN {X -30.656,Y -39.907,Z -123.482,A -90.000,B 90.000,C 0.000} C_DIS
LIN {X -30.749,Y -39.924,Z -123.161,A -90.000,B 90.000,C 0.000} C_DIS
LIN {X -30.796,Y -39.929,Z -122.991,A -90.000,B 90.000,C 0.000} C_DIS
LIN {X -30.917,Y -39.947,Z -122.567,A -90.000,B 90.000,C 0.000} C_DIS
LIN {X -30.992,Y -39.942,Z -122.393,A -90.000,B 90.000,C 0.000} C_DIS
LIN {X -31.477,Y -39.860,Z -121.227,A -90.000,B 90.000,C 0.000} C_DIS
LIN {X -31.526,Y -39.859,Z -121.117,A -90.000,B 90.000,C 0.000} C_DIS
LIN {X -31.620,Y -39.860,Z -120.882,A -90.000,B 90.000,C 0.000} C_DIS
LIN {X -31.779,Y -39.873,Z -120.422,A -90.000,B 90.000,C 0.000} C_DIS
LIN {X -31.846,Y -39.882,Z -120.205,A -90.000,B 90.000,C 0.000} C_DIS
LIN {X -31.907,Y -39.893,Z -119.991,A -90.000,B 90.000,C 0.000} C_DIS
LIN {X -32.006,Y -39.899,Z -119.622,A -90.000,B 90.000,C 0.000} C_DIS
LIN {X -32.055,Y -39.904,Z -119.428,A -90.000,B 90.000,C 0.000} C_DIS
LIN {X -32.207,Y -39.898,Z -118.791,A -90.000,B 90.000,C 0.000} C_DIS
LIN {X -32.248,Y -39.894,Z -118.615,A -90.000,B 90.000,C 0.000} C_DIS
LIN {X -32.532,Y -39.820,Z -117.856,A -90.000,B 90.000,C 0.000} C_DIS
LIN {X -32.573,Y -39.809,Z -117.750,A -90.000,B 90.000,C 0.000} C_DIS
LIN {X -32.704,Y -39.795,Z -117.431,A -90.000,B 90.000,C 0.000} C_DIS
LIN {X -32.951,Y -39.777,Z -116.785,A -90.000,B 90.000,C 0.000} C_DIS
LIN {X -33.070,Y -39.773,Z -116.445,A -90.000,B 90.000,C 0.000} C_DIS
LIN {X -33.138,Y -39.774,Z -116.228,A -90.000,B 90.000,C 0.000} C_DIS
LIN {X -33.204,Y -39.778,Z -115.983,A -90.000,B 90.000,C 0.000} C_DIS
LIN {X -33.290,Y -39.772,Z -115.630,A -90.000,B 90.000,C 0.000} C_DIS
LIN {X -33.310,Y -39.770,Z -115.531,A -90.000,B 90.000,C 0.000} C_DIS
LIN {X -33.354,Y -39.768,Z -115.296,A -90.000,B 90.000,C 0.000} C_DIS
LIN {X -33.404,Y -39.774,Z -114.936,A -90.000,B 90.000,C 0.000} C_DIS
LIN {X -33.498,Y -39.769,Z -114.186,A -90.000,B 90.000,C 0.000} C_DIS
LIN {X -33.515,Y -39.768,Z -114.049,A -90.000,B 90.000,C 0.000} C_DIS
LIN {X -33.553,Y -39.758,Z -113.866,A -90.000,B 90.000,C 0.000} C_DIS
LIN {X -33.659,Y -39.753,Z -113.397,A -90.000,B 90.000,C 0.000} C_DIS
LIN {X -33.700,Y -39.755,Z -113.180,A -90.000,B 90.000,C 0.000} C_DIS
LIN {X -33.718,Y -39.758,Z -113.064,A -90.000,B 90.000,C 0.000} C_DIS
LIN {X -33.757,Y -39.756,Z -112.760,A -90.000,B 90.000,C 0.000} C_DIS
LIN {X -33.775,Y -39.756,Z -112.578,A -90.000,B 90.000,C 0.000} C_DIS
LIN {X -33.817,Y -39.749,Z -112.076,A -90.000,B 90.000,C 0.000} C_DIS
LIN {X -33.852,Y -39.752,Z -111.742,A -90.000,B 90.000,C 0.000} C_DIS
LIN {X -33.926,Y -39.745,Z -111.265,A -90.000,B 90.000,C 0.000} C_DIS
LIN {X -34.067,Y -39.715,Z -110.315,A -90.000,B 90.000,C 0.000} C_DIS
LIN {X -34.101,Y -39.704,Z -110.035,A -90.000,B 90.000,C 0.000} C_DIS
LIN {X -34.124,Y -39.690,Z -109.802,A -90.000,B 90.000,C 0.000} C_DIS
LIN {X -34.140,Y -39.661,Z -109.446,A -90.000,B 90.000,C 0.000} C_DIS
LIN {X -34.147,Y -39.647,Z -109.276,A -90.000,B 90.000,C 0.000} C_DIS
LIN {X -34.146,Y -39.636,Z -109.080,A -90.000,B 90.000,C 0.000} C_DIS
LIN {X -34.142,Y -39.631,Z -108.952,A -90.000,B 90.000,C 0.000} C_DIS
LIN {X -34.122,Y -39.623,Z -108.599,A -90.000,B 90.000,C 0.000} C_DIS
LIN {X -34.090,Y -39.617,Z -108.164,A -90.000,B 90.000,C 0.000} C_DIS
LIN {X -34.028,Y -39.623,Z -107.156,A -90.000,B 90.000,C 0.000} C_DIS
LIN {X -34.013,Y -39.615,Z -106.829,A -90.000,B 90.000,C 0.000} C_DIS
LIN {X -33.993,Y -39.598,Z -106.510,A -90.000,B 90.000,C 0.000} C_DIS
LIN {X -33.979,Y -39.590,Z -106.327,A -90.000,B 90.000,C 0.000} C_DIS
LIN {X -33.949,Y -39.583,Z -106.016,A -90.000,B 90.000,C 0.000} C_DIS
LIN {X -33.895,Y -39.573,Z -105.452,A -90.000,B 90.000,C 0.000} C_DIS
LIN {X -33.869,Y -39.568,Z -105.165,A -90.000,B 90.000,C 0.000} C_DIS
LIN {X -33.861,Y -39.565,Z -105.071,A -90.000,B 90.000,C 0.000} C_DIS
LIN {X -33.789,Y -39.517,Z -104.304,A -90.000,B 90.000,C 0.000} C_DIS
LIN {X -33.731,Y -39.474,Z -103.767,A -90.000,B 90.000,C 0.000} C_DIS
LIN {X -33.686,Y -39.441,Z -103.418,A -90.000,B 90.000,C 0.000} C_DIS
LIN {X -33.616,Y -39.378,Z -102.809,A -90.000,B 90.000,C 0.000} C_DIS
LIN {X -33.592,Y -39.361,Z -102.627,A -90.000,B 90.000,C 0.000} C_DIS
LIN {X -33.483,Y -39.308,Z -101.863,A -90.000,B 90.000,C 0.000} C_DIS
LIN {X -33.483,Y -60.000,Z -101.863,A -90.000,B 90.000,C 0.000} C_DIS
LIN {X -82.090,Y -60.000,Z -243.561,A -90.000,B 90.000,C 0.000} C_DIS
LIN {X -82.090,Y -39.992,Z -243.561,A -90.000,B 90.000,C 0.000} C_DIS
LIN {X -82.077,Y -39.956,Z -243.491,A -90.000,B 90.000,C 0.000} C_DIS
LIN {X -82.054,Y -39.908,Z -243.396,A -90.000,B 90.000,C 0.000} C_DIS
LIN {X -81.980,Y -39.773,Z -243.118,A -90.000,B 90.000,C 0.000} C_DIS
LIN {X -81.942,Y -39.721,Z -243.007,A -90.000,B 90.000,C 0.000} C_DIS
LIN {X -81.865,Y -39.631,Z -242.804,A -90.000,B 90.000,C 0.000} C_DIS
LIN {X -81.810,Y -39.578,Z -242.680,A -90.000,B 90.000,C 0.000} C_DIS
LIN {X -81.767,Y -39.541,Z -242.588,A -90.000,B 90.000,C 0.000} C_DIS
LIN {X -81.688,Y -39.480,Z -242.437,A -90.000,B 90.000,C 0.000} C_DIS
LIN {X -81.592,Y -39.417,Z -242.274,A -90.000,B 90.000,C 0.000} C_DIS
LIN {X -81.388,Y -39.308,Z -241.971,A -90.000,B 90.000,C 0.000} C_DIS
LIN {X -81.318,Y -39.274,Z -241.864,A -90.000,B 90.000,C 0.000} C_DIS
LIN {X -81.236,Y -39.220,Z -241.726,A -90.000,B 90.000,C 0.000} C_DIS
LIN {X -81.196,Y -39.188,Z -241.647,A -90.000,B 90.000,C 0.000} C_DIS
LIN {X -81.155,Y -39.144,Z -241.549,A -90.000,B 90.000,C 0.000} C_DIS
LIN {X -81.140,Y -39.117,Z -241.496,A -90.000,B 90.000,C 0.000} C_DIS
LIN {X -81.136,Y -39.104,Z -241.473,A -90.000,B 90.000,C 0.000} C_DIS
LIN {X -81.136,Y -39.081,Z -241.434,A -90.000,B 90.000,C 0.000} C_DIS
LIN {X -81.145,Y -39.060,Z -241.404,A -90.000,B 90.000,C 0.000} C_DIS
LIN {X -81.153,Y -39.050,Z -241.393,A -90.000,B 90.000,C 0.000} C_DIS
LIN {X -81.175,Y -39.032,Z -241.376,A -90.000,B 90.000,C 0.000} C_DIS
LIN {X -81.206,Y -39.016,Z -241.367,A -90.000,B 90.000,C 0.000} C_DIS
LIN {X -81.244,Y -39.002,Z -241.367,A -90.000,B 90.000,C 0.000} C_DIS
LIN {X -81.289,Y -38.989,Z -241.374,A -90.000,B 90.000,C 0.000} C_DIS
LIN {X -81.341,Y -38.979,Z -241.388,A -90.000,B 90.000,C 0.000} C_DIS
LIN {X -81.400,Y -38.970,Z -241.408,A -90.000,B 90.000,C 0.000} C_DIS
LIN {X -81.465,Y -38.963,Z -241.436,A -90.000,B 90.000,C 0.000} C_DIS
LIN {X -81.612,Y -38.953,Z -241.508,A -90.000,B 90.000,C 0.000} C_DIS
LIN {X -81.778,Y -38.949,Z -241.603,A -90.000,B 90.000,C 0.000} C_DIS
LIN {X -81.962,Y -38.951,Z -241.716,A -90.000,B 90.000,C 0.000} C_DIS
LIN {X -82.158,Y -38.957,Z -241.846,A -90.000,B 90.000,C 0.000} C_DIS
LIN {X -82.471,Y -38.975,Z -242.064,A -90.000,B 90.000,C 0.000} C_DIS
LIN {X -82.795,Y -38.999,Z -242.304,A -90.000,B 90.000,C 0.000} C_DIS
LIN {X -83.013,Y -39.016,Z -242.470,A -90.000,B 90.000,C 0.000} C_DIS
LIN {X -83.228,Y -39.036,Z -242.639,A -90.000,B 90.000,C 0.000} C_DIS
LIN {X -83.437,Y -39.057,Z -242.808,A -90.000,B 90.000,C 0.000} C_DIS
LIN {X -83.637,Y -39.080,Z -242.973,A -90.000,B 90.000,C 0.000} C_DIS
LIN {X -83.824,Y -39.104,Z -243.132,A -90.000,B 90.000,C 0.000} C_DIS
LIN {X -84.075,Y -39.141,Z -243.353,A -90.000,B 90.000,C 0.000} C_DIS
LIN {X -84.280,Y -39.178,Z -243.546,A -90.000,B 90.000,C 0.000} C_DIS
LIN {X -84.428,Y -39.214,Z -243.699,A -90.000,B 90.000,C 0.000} C_DIS
LIN {X -84.490,Y -39.236,Z -243.776,A -90.000,B 90.000,C 0.000} C_DIS
LIN {X -84.509,Y -39.246,Z -243.805,A -90.000,B 90.000,C 0.000} C_DIS
LIN {X -84.520,Y -39.260,Z -243.837,A -90.000,B 90.000,C 0.000} C_DIS
LIN {X -84.516,Y -39.269,Z -243.850,A -90.000,B 90.000,C 0.000} C_DIS
LIN {X -84.511,Y -39.273,Z -243.853,A -90.000,B 90.000,C 0.000} C_DIS
LIN {X -84.492,Y -39.281,Z -243.855,A -90.000,B 90.000,C 0.000} C_DIS
LIN {X -84.479,Y -39.285,Z -243.853,A -90.000,B 90.000,C 0.000} C_DIS
LIN {X -84.445,Y -39.292,Z -243.843,A -90.000,B 90.000,C 0.000} C_DIS
LIN {X -84.373,Y -39.301,Z -243.813,A -90.000,B 90.000,C 0.000} C_DIS
LIN {X -84.310,Y -39.305,Z -243.781,A -90.000,B 90.000,C 0.000} C_DIS
LIN {X -84.150,Y -39.312,Z -243.691,A -90.000,B 90.000,C 0.000} C_DIS
LIN {X -84.050,Y -39.314,Z -243.631,A -90.000,B 90.000,C 0.000} C_DIS
LIN {X -83.938,Y -39.308,Z -243.561,A -90.000,B 90.000,C 0.000} C_DIS
LIN {X -82.050,Y -39.308,Z -242.371,A -90.000,B 90.000,C 0.000} C_DIS
LIN {X -79.673,Y -39.308,Z -240.934,A -90.000,B 90.000,C 0.000} C_DIS
LIN {X -73.869,Y -39.308,Z -237.553,A -90.000,B 90.000,C 0.000} C_DIS
LIN {X -73.538,Y -39.308,Z -237.369,A -90.000,B 90.000,C 0.000} C_DIS
LIN {X -72.765,Y -39.308,Z -236.944,A -90.000,B 90.000,C 0.000} C_DIS
LIN {X -69.296,Y -39.308,Z -235.057,A -90.000,B 90.000,C 0.000} C_DIS
LIN {X -66.594,Y -39.308,Z -233.591,A -90.000,B 90.000,C 0.000} C_DIS
LIN {X -65.340,Y -39.308,Z -232.926,A -90.000,B 90.000,C 0.000} C_DIS
LIN {X -62.891,Y -39.308,Z -231.680,A -90.000,B 90.000,C 0.000} C_DIS
LIN {X -56.747,Y -39.308,Z -228.550,A -90.000,B 90.000,C 0.000} C_DIS
LIN {X -48.418,Y -39.308,Z -224.423,A -90.000,B 90.000,C 0.000} C_DIS
LIN {X -42.976,Y -39.308,Z -221.766,A -90.000,B 90.000,C 0.000} C_DIS
LIN {X -40.571,Y -39.308,Z -220.601,A -90.000,B 90.000,C 0.000} C_DIS
LIN {X -33.530,Y -39.308,Z -217.129,A -90.000,B 90.000,C 0.000} C_DIS
LIN {X -33.084,Y -39.308,Z -216.900,A -90.000,B 90.000,C 0.000} C_DIS
LIN {X -31.983,Y -39.308,Z -216.327,A -90.000,B 90.000,C 0.000} C_DIS
LIN {X -28.842,Y -39.308,Z -214.764,A -90.000,B 90.000,C 0.000} C_DIS
LIN {X -27.499,Y -39.308,Z -214.089,A -90.000,B 90.000,C 0.000} C_DIS
LIN {X -25.145,Y -39.308,Z -212.832,A -90.000,B 90.000,C 0.000} C_DIS
LIN {X -22.635,Y -39.308,Z -211.454,A -90.000,B 90.000,C 0.000} C_DIS
LIN {X -21.586,Y -39.308,Z -210.840,A -90.000,B 90.000,C 0.000} C_DIS
LIN {X -18.141,Y -39.308,Z -208.758,A -90.000,B 90.000,C 0.000} C_DIS
LIN {X -15.583,Y -39.308,Z -207.084,A -90.000,B 90.000,C 0.000} C_DIS
LIN {X -14.619,Y -39.308,Z -206.475,A -90.000,B 90.000,C 0.000} C_DIS
LIN {X -14.349,Y -39.308,Z -206.298,A -90.000,B 90.000,C 0.000} C_DIS
LIN {X -13.901,Y -39.308,Z -205.987,A -90.000,B 90.000,C 0.000} C_DIS
LIN {X -10.422,Y -39.308,Z -203.579,A -90.000,B 90.000,C 0.000} C_DIS
LIN {X -8.882,Y -39.308,Z -202.422,A -90.000,B 90.000,C 0.000} C_DIS
LIN {X -6.639,Y -39.308,Z -200.746,A -90.000,B 90.000,C 0.000} C_DIS
LIN {X -4.318,Y -39.308,Z -198.867,A -90.000,B 90.000,C 0.000} C_DIS
LIN {X -3.070,Y -39.308,Z -197.866,A -90.000,B 90.000,C 0.000} C_DIS
LIN {X -0.285,Y -39.308,Z -195.431,A -90.000,B 90.000,C 0.000} C_DIS
LIN {X 0.445,Y -39.308,Z -194.809,A -90.000,B 90.000,C 0.000} C_DIS
LIN {X 1.053,Y -39.308,Z -194.268,A -90.000,B 90.000,C 0.000} C_DIS
LIN {X 4.059,Y -39.308,Z -191.417,A -90.000,B 90.000,C 0.000} C_DIS
LIN {X 4.362,Y -39.308,Z -191.137,A -90.000,B 90.000,C 0.000} C_DIS
LIN {X 7.587,Y -39.308,Z -187.942,A -90.000,B 90.000,C 0.000} C_DIS
LIN {X 10.879,Y -39.308,Z -184.628,A -90.000,B 90.000,C 0.000} C_DIS
LIN {X 13.412,Y -39.308,Z -182.108,A -90.000,B 90.000,C 0.000} C_DIS
LIN {X 13.850,Y -39.308,Z -181.643,A -90.000,B 90.000,C 0.000} C_DIS
LIN {X 14.756,Y -39.308,Z -180.753,A -90.000,B 90.000,C 0.000} C_DIS
LIN {X 16.722,Y -39.308,Z -178.878,A -90.000,B 90.000,C 0.000} C_DIS
LIN {X 17.427,Y -39.308,Z -178.218,A -90.000,B 90.000,C 0.000} C_DIS
LIN {X 19.806,Y -39.308,Z -176.001,A -90.000,B 90.000,C 0.000} C_DIS
LIN {X 21.099,Y -39.308,Z -174.778,A -90.000,B 90.000,C 0.000} C_DIS
LIN {X 21.775,Y -39.308,Z -174.116,A -90.000,B 90.000,C 0.000} C_DIS
LIN {X 22.710,Y -39.308,Z -173.175,A -90.000,B 90.000,C 0.000} C_DIS
LIN {X 23.592,Y -39.308,Z -172.209,A -90.000,B 90.000,C 0.000} C_DIS
LIN {X 24.398,Y -39.308,Z -171.299,A -90.000,B 90.000,C 0.000} C_DIS
LIN {X 24.751,Y -39.308,Z -170.869,A -90.000,B 90.000,C 0.000} C_DIS
LIN {X 25.795,Y -39.308,Z -169.569,A -90.000,B 90.000,C 0.000} C_DIS
LIN {X 26.363,Y -39.308,Z -168.818,A -90.000,B 90.000,C 0.000} C_DIS
LIN {X 27.304,Y -39.308,Z -167.549,A -90.000,B 90.000,C 0.000} C_DIS
LIN {X 27.908,Y -39.308,Z -166.698,A -90.000,B 90.000,C 0.000} C_DIS
LIN {X 28.781,Y -39.308,Z -165.453,A -90.000,B 90.000,C 0.000} C_DIS
LIN {X 30.270,Y -39.308,Z -163.269,A -90.000,B 90.000,C 0.000} C_DIS
LIN {X 30.883,Y -39.308,Z -162.317,A -90.000,B 90.000,C 0.000} C_DIS
LIN {X 31.523,Y -39.308,Z -161.328,A -90.000,B 90.000,C 0.000} C_DIS
LIN {X 31.840,Y -39.308,Z -160.784,A -90.000,B 90.000,C 0.000} C_DIS
LIN {X 32.627,Y -39.308,Z -159.456,A -90.000,B 90.000,C 0.000} C_DIS
LIN {X 32.756,Y -39.308,Z -159.206,A -90.000,B 90.000,C 0.000} C_DIS
LIN {X 33.059,Y -39.308,Z -158.636,A -90.000,B 90.000,C 0.000} C_DIS
LIN {X 33.401,Y -39.308,Z -157.905,A -90.000,B 90.000,C 0.000} C_DIS
LIN {X 33.535,Y -39.308,Z -157.623,A -90.000,B 90.000,C 0.000} C_DIS
LIN {X 33.768,Y -39.308,Z -156.986,A -90.000,B 90.000,C 0.000} C_DIS
LIN {X 33.887,Y -39.308,Z -156.691,A -90.000,B 90.000,C 0.000} C_DIS
LIN {X 34.030,Y -39.308,Z -156.021,A -90.000,B 90.000,C 0.000} C_DIS
LIN {X 34.061,Y -39.308,Z -155.879,A -90.000,B 90.000,C 0.000} C_DIS
LIN {X 34.205,Y -39.308,Z -155.398,A -90.000,B 90.000,C 0.000} C_DIS
LIN {X 34.183,Y -39.308,Z -155.049,A -90.000,B 90.000,C 0.000} C_DIS
LIN {X 34.203,Y -39.308,Z -154.813,A -90.000,B 90.000,C 0.000} C_DIS
LIN {X 34.263,Y -39.308,Z -154.346,A -90.000,B 90.000,C 0.000} C_DIS
LIN {X 34.105,Y -39.308,Z -154.193,A -90.000,B 90.000,C 0.000} C_DIS
LIN {X 34.004,Y -39.308,Z -154.051,A -90.000,B 90.000,C 0.000} C_DIS
LIN {X 33.813,Y -39.308,Z -153.554,A -90.000,B 90.000,C 0.000} C_DIS
LIN {X 32.681,Y -39.308,Z -153.424,A -90.000,B 90.000,C 0.000} C_DIS
LIN {X 32.497,Y -39.308,Z -153.346,A -90.000,B 90.000,C 0.000} C_DIS
LIN {X 32.282,Y -39.308,Z -153.385,A -90.000,B 90.000,C 0.000} C_DIS
LIN {X 32.139,Y -39.308,Z -153.408,A -90.000,B 90.000,C 0.000} C_DIS
LIN {X 31.179,Y -39.308,Z -153.506,A -90.000,B 90.000,C 0.000} C_DIS
LIN {X 30.480,Y -39.308,Z -153.689,A -90.000,B 90.000,C 0.000} C_DIS
LIN {X 30.302,Y -39.308,Z -153.717,A -90.000,B 90.000,C 0.000} C_DIS
LIN {X 29.690,Y -39.308,Z -153.718,A -90.000,B 90.000,C 0.000} C_DIS
LIN {X 28.375,Y -39.308,Z -153.888,A -90.000,B 90.000,C 0.000} C_DIS
LIN {X 28.117,Y -39.308,Z -153.858,A -90.000,B 90.000,C 0.000} C_DIS
LIN {X 28.088,Y -39.308,Z -153.853,A -90.000,B 90.000,C 0.000} C_DIS
LIN {X 27.923,Y -39.308,Z -153.783,A -90.000,B 90.000,C 0.000} C_DIS
LIN {X 27.783,Y -39.308,Z -153.671,A -90.000,B 90.000,C 0.000} C_DIS
LIN {X 27.757,Y -39.308,Z -153.634,A -90.000,B 90.000,C 0.000} C_DIS
LIN {X 26.945,Y -39.308,Z -152.621,A -90.000,B 90.000,C 0.000} C_DIS
LIN {X 26.842,Y -39.308,Z -152.475,A -90.000,B 90.000,C 0.000} C_DIS
LIN {X 26.782,Y -39.308,Z -152.306,A -90.000,B 90.000,C 0.000} C_DIS
LIN {X 26.771,Y -39.308,Z -152.097,A -90.000,B 90.000,C 0.000} C_DIS
LIN {X 26.770,Y -39.308,Z -152.015,A -90.000,B 90.000,C 0.000} C_DIS
LIN {X 27.127,Y -39.308,Z -150.418,A -90.000,B 90.000,C 0.000} C_DIS
LIN {X 27.294,Y -39.308,Z -149.727,A -90.000,B 90.000,C 0.000} C_DIS
LIN {X 27.682,Y -39.308,Z -148.754,A -90.000,B 90.000,C 0.000} C_DIS
LIN {X 27.852,Y -39.308,Z -148.436,A -90.000,B 90.000,C 0.000} C_DIS
LIN {X 27.967,Y -39.308,Z -148.229,A -90.000,B 90.000,C 0.000} C_DIS
LIN {X 28.144,Y -39.308,Z -147.930,A -90.000,B 90.000,C 0.000} C_DIS
LIN {X 30.465,Y -39.308,Z -145.075,A -90.000,B 90.000,C 0.000} C_DIS
LIN {X 30.620,Y -39.308,Z -144.897,A -90.000,B 90.000,C 0.000} C_DIS
LIN {X 33.046,Y -39.308,Z -142.494,A -90.000,B 90.000,C 0.000} C_DIS
LIN {X 33.252,Y -39.308,Z -142.296,A -90.000,B 90.000,C 0.000} C_DIS
LIN {X 36.292,Y -39.308,Z -139.650,A -90.000,B 90.000,C 0.000} C_DIS
LIN {X 39.047,Y -39.308,Z -137.332,A -90.000,B 90.000,C 0.000} C_DIS
LIN {X 39.105,Y -39.308,Z -137.277,A -90.000,B 90.000,C 0.000} C_DIS
LIN {X 42.001,Y -39.308,Z -134.723,A -90.000,B 90.000,C 0.000} C_DIS
LIN {X 42.573,Y -39.308,Z -134.122,A -90.000,B 90.000,C 0.000} C_DIS
LIN {X 44.563,Y -39.308,Z -132.039,A -90.000,B 90.000,C 0.000} C_DIS
LIN {X 44.654,Y -39.308,Z -131.919,A -90.000,B 90.000,C 0.000} C_DIS
LIN {X 44.910,Y -39.308,Z -131.620,A -90.000,B 90.000,C 0.000} C_DIS
LIN {X 44.046,Y -39.308,Z -132.330,A -90.000,B 90.000,C 0.000} C_DIS
LIN {X 43.764,Y -39.308,Z -132.546,A -90.000,B 90.000,C 0.000} C_DIS
LIN {X 41.244,Y -39.308,Z -134.370,A -90.000,B 90.000,C 0.000} C_DIS
LIN {X 40.433,Y -39.308,Z -134.947,A -90.000,B 90.000,C 0.000} C_DIS
LIN {X 39.136,Y -39.308,Z -135.810,A -90.000,B 90.000,C 0.000} C_DIS
LIN {X 37.125,Y -39.308,Z -137.175,A -90.000,B 90.000,C 0.000} C_DIS
LIN {X 36.392,Y -39.308,Z -137.690,A -90.000,B 90.000,C 0.000} C_DIS
LIN {X 34.951,Y -39.308,Z -138.691,A -90.000,B 90.000,C 0.000} C_DIS
LIN {X 30.879,Y -39.308,Z -141.427,A -90.000,B 90.000,C 0.000} C_DIS
LIN {X 30.646,Y -39.308,Z -141.575,A -90.000,B 90.000,C 0.000} C_DIS
LIN {X 27.391,Y -39.308,Z -143.580,A -90.000,B 90.000,C 0.000} C_DIS
LIN {X 27.076,Y -39.308,Z -143.769,A -90.000,B 90.000,C 0.000} C_DIS
LIN {X 26.469,Y -39.308,Z -144.092,A -90.000,B 90.000,C 0.000} C_DIS
LIN {X 23.452,Y -39.308,Z -145.710,A -90.000,B 90.000,C 0.000} C_DIS
LIN {X 23.202,Y -39.308,Z -145.837,A -90.000,B 90.000,C 0.000} C_DIS
LIN {X 22.804,Y -39.308,Z -146.028,A -90.000,B 90.000,C 0.000} C_DIS
LIN {X 21.536,Y -39.308,Z -146.592,A -90.000,B 90.000,C 0.000} C_DIS
LIN {X 19.654,Y -39.308,Z -147.362,A -90.000,B 90.000,C 0.000} C_DIS
LIN {X 18.722,Y -39.308,Z -147.733,A -90.000,B 90.000,C 0.000} C_DIS
LIN {X 18.322,Y -39.308,Z -147.870,A -90.000,B 90.000,C 0.000} C_DIS
LIN {X 15.456,Y -39.308,Z -148.767,A -90.000,B 90.000,C 0.000} C_DIS
LIN {X 13.379,Y -39.308,Z -149.397,A -90.000,B 90.000,C 0.000} C_DIS
LIN {X 12.982,Y -39.308,Z -149.507,A -90.000,B 90.000,C 0.000} C_DIS
LIN {X 10.590,Y -39.308,Z -150.021,A -90.000,B 90.000,C 0.000} C_DIS
LIN {X 8.962,Y -39.308,Z -150.342,A -90.000,B 90.000,C 0.000} C_DIS
LIN {X 8.697,Y -39.308,Z -150.392,A -90.000,B 90.000,C 0.000} C_DIS
LIN {X 8.242,Y -39.308,Z -150.461,A -90.000,B 90.000,C 0.000} C_DIS
LIN {X 5.051,Y -39.308,Z -150.791,A -90.000,B 90.000,C 0.000} C_DIS
LIN {X 4.632,Y -39.308,Z -150.819,A -90.000,B 90.000,C 0.000} C_DIS
LIN {X 3.504,Y -39.308,Z -150.807,A -90.000,B 90.000,C 0.000} C_DIS
LIN {X 1.445,Y -39.308,Z -150.775,A -90.000,B 90.000,C 0.000} C_DIS
LIN {X 1.128,Y -39.308,Z -150.763,A -90.000,B 90.000,C 0.000} C_DIS
LIN {X 0.705,Y -39.308,Z -150.742,A -90.000,B 90.000,C 0.000} C_DIS
LIN {X -2.262,Y -39.308,Z -150.289,A -90.000,B 90.000,C 0.000} C_DIS
LIN {X -3.175,Y -39.308,Z -150.137,A -90.000,B 90.000,C 0.000} C_DIS
LIN {X -3.263,Y -39.308,Z -150.120,A -90.000,B 90.000,C 0.000} C_DIS
LIN {X -3.401,Y -39.308,Z -150.083,A -90.000,B 90.000,C 0.000} C_DIS
LIN {X -6.981,Y -39.308,Z -149.070,A -90.000,B 90.000,C 0.000} C_DIS
LIN {X -7.213,Y -39.308,Z -149.002,A -90.000,B 90.000,C 0.000} C_DIS
LIN {X -7.391,Y -39.308,Z -148.937,A -90.000,B 90.000,C 0.000} C_DIS
LIN {X -10.888,Y -39.308,Z -147.493,A -90.000,B 90.000,C 0.000} C_DIS
LIN {X -11.273,Y -39.308,Z -147.329,A -90.000,B 90.000,C 0.000} C_DIS
LIN {X -14.840,Y -39.308,Z -145.346,A -90.000,B 90.000,C 0.000} C_DIS
LIN {X -15.208,Y -39.308,Z -145.135,A -90.000,B 90.000,C 0.000} C_DIS
LIN {X -16.699,Y -39.308,Z -144.089,A -90.000,B 90.000,C 0.000} C_DIS
LIN {X -18.639,Y -39.308,Z -142.735,A -90.000,B 90.000,C 0.000} C_DIS
LIN {X -18.979,Y -39.308,Z -142.483,A -90.000,B 90.000,C 0.000} C_DIS
LIN {X -19.638,Y -39.308,Z -141.926,A -90.000,B 90.000,C 0.000} C_DIS
LIN {X -21.470,Y -39.308,Z -140.297,A -90.000,B 90.000,C 0.000} C_DIS
LIN {X -21.859,Y -39.308,Z -139.933,A -90.000,B 90.000,C 0.000} C_DIS
LIN {X -22.086,Y -39.308,Z -139.717,A -90.000,B 90.000,C 0.000} C_DIS
LIN {X -22.365,Y -39.308,Z -139.426,A -90.000,B 90.000,C 0.000} C_DIS
LIN {X -23.764,Y -39.308,Z -137.843,A -90.000,B 90.000,C 0.000} C_DIS
LIN {X -24.931,Y -39.308,Z -136.495,A -90.000,B 90.000,C 0.000} C_DIS
LIN {X -25.172,Y -39.308,Z -136.173,A -90.000,B 90.000,C 0.000} C_DIS
LIN {X -26.004,Y -39.308,Z -135.031,A -90.000,B 90.000,C 0.000} C_DIS
LIN {X -27.151,Y -39.308,Z -133.417,A -90.000,B 90.000,C 0.000} C_DIS
LIN {X -27.305,Y -39.308,Z -133.179,A -90.000,B 90.000,C 0.000} C_DIS
LIN {X -28.053,Y -39.308,Z -131.806,A -90.000,B 90.000,C 0.000} C_DIS
LIN {X -28.216,Y -39.308,Z -131.495,A -90.000,B 90.000,C 0.000} C_DIS
LIN {X -29.086,Y -39.308,Z -129.803,A -90.000,B 90.000,C 0.000} C_DIS
LIN {X -29.842,Y -39.308,Z -128.248,A -90.000,B 90.000,C 0.000} C_DIS
LIN {X -30.482,Y -39.308,Z -126.862,A -90.000,B 90.000,C 0.000} C_DIS
LIN {X -31.238,Y -39.308,Z -125.138,A -90.000,B 90.000,C 0.000} C_DIS
LIN {X -31.576,Y -39.308,Z -124.254,A -90.000,B 90.000,C 0.000} C_DIS
LIN {X -31.639,Y -39.308,Z -124.078,A -90.000,B 90.000,C 0.000} C_DIS
LIN {X -31.695,Y -39.308,Z -123.911,A -90.000,B 90.000,C 0.000} C_DIS
LIN {X -32.007,Y -39.308,Z -122.862,A -90.000,B 90.000,C 0.000} C_DIS
LIN {X -32.505,Y -39.308,Z -121.652,A -90.000,B 90.000,C 0.000} C_DIS
LIN {X -32.622,Y -39.308,Z -121.324,A -90.000,B 90.000,C 0.000} C_DIS
LIN {X -32.665,Y -39.308,Z -121.190,A -90.000,B 90.000,C 0.000} C_DIS
LIN {X -32.970,Y -39.308,Z -119.786,A -90.000,B 90.000,C 0.000} C_DIS
LIN {X -33.393,Y -39.308,Z -118.524,A -90.000,B 90.000,C 0.000} C_DIS
LIN {X -33.496,Y -39.308,Z -118.063,A -90.000,B 90.000,C 0.000} C_DIS
LIN {X -33.745,Y -39.308,Z -117.219,A -90.000,B 90.000,C 0.000} C_DIS
LIN {X -33.815,Y -39.308,Z -116.875,A -90.000,B 90.000,C 0.000} C_DIS
LIN {X -34.023,Y -39.308,Z -115.796,A -90.000,B 90.000,C 0.000} C_DIS
LIN {X -34.104,Y -39.308,Z -115.407,A -90.000,B 90.000,C 0.000} C_DIS
LIN {X -34.129,Y -39.308,Z -115.287,A -90.000,B 90.000,C 0.000} C_DIS
LIN {X -34.255,Y -39.308,Z -114.181,A -90.000,B 90.000,C 0.000} C_DIS
LIN {X -34.574,Y -39.308,Z -112.661,A -90.000,B 90.000,C 0.000} C_DIS
LIN {X -34.644,Y -39.308,Z -112.317,A -90.000,B 90.000,C 0.000} C_DIS
LIN {X -34.650,Y -39.308,Z -112.254,A -90.000,B 90.000,C 0.000} C_DIS
LIN {X -34.670,Y -39.308,Z -111.910,A -90.000,B 90.000,C 0.000} C_DIS
LIN {X -34.679,Y -39.308,Z -110.709,A -90.000,B 90.000,C 0.000} C_DIS
LIN {X -34.671,Y -39.308,Z -110.093,A -90.000,B 90.000,C 0.000} C_DIS
LIN {X -34.685,Y -39.308,Z -109.756,A -90.000,B 90.000,C 0.000} C_DIS
LIN {X -34.686,Y -39.308,Z -109.289,A -90.000,B 90.000,C 0.000} C_DIS
LIN {X -34.656,Y -39.308,Z -108.938,A -90.000,B 90.000,C 0.000} C_DIS
LIN {X -34.605,Y -39.308,Z -108.390,A -90.000,B 90.000,C 0.000} C_DIS
LIN {X -34.518,Y -39.308,Z -106.749,A -90.000,B 90.000,C 0.000} C_DIS
LIN {X -34.487,Y -39.308,Z -106.399,A -90.000,B 90.000,C 0.000} C_DIS
LIN {X -34.168,Y -39.308,Z -104.674,A -90.000,B 90.000,C 0.000} C_DIS
LIN {X -34.078,Y -39.308,Z -104.267,A -90.000,B 90.000,C 0.000} C_DIS
LIN {X -34.044,Y -39.308,Z -104.094,A -90.000,B 90.000,C 0.000} C_DIS
LIN {X -33.676,Y -39.308,Z -102.672,A -90.000,B 90.000,C 0.000} C_DIS
LIN {X -33.475,Y -39.308,Z -101.829,A -90.000,B 90.000,C 0.000} C_DIS
LIN {X -33.295,Y -39.308,Z -101.115,A -90.000,B 90.000,C 0.000} C_DIS
LIN {X -32.985,Y -39.308,Z -99.770,A -90.000,B 90.000,C 0.000} C_DIS
LIN {X -32.917,Y -39.308,Z -99.521,A -90.000,B 90.000,C 0.000} C_DIS
LIN {X -32.442,Y -39.308,Z -97.882,A -90.000,B 90.000,C 0.000} C_DIS
LIN {X -32.324,Y -39.308,Z -97.490,A -90.000,B 90.000,C 0.000} C_DIS
LIN {X -32.271,Y -39.308,Z -97.295,A -90.000,B 90.000,C 0.000} C_DIS
LIN {X -32.023,Y -39.308,Z -96.531,A -90.000,B 90.000,C 0.000} C_DIS
LIN {X -31.737,Y -39.308,Z -95.546,A -90.000,B 90.000,C 0.000} C_DIS
LIN {X -31.582,Y -39.308,Z -95.030,A -90.000,B 90.000,C 0.000} C_DIS
LIN {X -31.476,Y -39.308,Z -94.700,A -90.000,B 90.000,C 0.000} C_DIS
LIN {X -31.055,Y -39.308,Z -93.522,A -90.000,B 90.000,C 0.000} C_DIS
LIN {X -30.857,Y -39.308,Z -92.865,A -90.000,B 90.000,C 0.000} C_DIS
LIN {X -30.743,Y -39.308,Z -92.504,A -90.000,B 90.000,C 0.000} C_DIS
LIN {X -30.667,Y -39.308,Z -92.302,A -90.000,B 90.000,C 0.000} C_DIS
LIN {X -30.460,Y -39.308,Z -91.632,A -90.000,B 90.000,C 0.000} C_DIS
LIN {X -30.200,Y -39.308,Z -90.856,A -90.000,B 90.000,C 0.000} C_DIS
LIN {X -30.126,Y -39.308,Z -90.503,A -90.000,B 90.000,C 0.000} C_DIS
LIN {X -30.129,Y -39.308,Z -90.390,A -90.000,B 90.000,C 0.000} C_DIS
LIN {X -30.109,Y -39.308,Z -90.155,A -90.000,B 90.000,C 0.000} C_DIS
LIN {X -29.809,Y -39.308,Z -88.740,A -90.000,B 90.000,C 0.000} C_DIS
LIN {X -29.635,Y -39.308,Z -87.958,A -90.000,B 90.000,C 0.000} C_DIS
LIN {X -29.621,Y -39.308,Z -87.909,A -90.000,B 90.000,C 0.000} C_DIS
LIN {X -29.616,Y -39.308,Z -87.866,A -90.000,B 90.000,C 0.000} C_DIS
LIN {X -29.577,Y -39.308,Z -87.691,A -90.000,B 90.000,C 0.000} C_DIS
LIN {X -29.491,Y -39.308,Z -87.533,A -90.000,B 90.000,C 0.000} C_DIS
LIN {X -29.319,Y -39.308,Z -87.262,A -90.000,B 90.000,C 0.000} C_DIS
LIN {X -29.231,Y -39.308,Z -87.119,A -90.000,B 90.000,C 0.000} C_DIS
LIN {X -28.770,Y -39.308,Z -86.279,A -90.000,B 90.000,C 0.000} C_DIS
LIN {X -28.582,Y -39.308,Z -85.950,A -90.000,B 90.000,C 0.000} C_DIS
LIN {X -28.356,Y -39.308,Z -85.551,A -90.000,B 90.000,C 0.000} C_DIS
LIN {X -28.200,Y -39.308,Z -85.373,A -90.000,B 90.000,C 0.000} C_DIS
LIN {X -27.668,Y -39.308,Z -84.818,A -90.000,B 90.000,C 0.000} C_DIS
LIN {X -27.271,Y -39.308,Z -84.430,A -90.000,B 90.000,C 0.000} C_DIS
LIN {X -27.205,Y -39.308,Z -84.342,A -90.000,B 90.000,C 0.000} C_DIS
LIN {X -26.561,Y -39.308,Z -83.543,A -90.000,B 90.000,C 0.000} C_DIS
LIN {X -26.360,Y -39.308,Z -83.328,A -90.000,B 90.000,C 0.000} C_DIS
LIN {X -25.889,Y -39.308,Z -82.877,A -90.000,B 90.000,C 0.000} C_DIS
LIN {X -24.943,Y -39.308,Z -81.775,A -90.000,B 90.000,C 0.000} C_DIS
LIN {X -24.594,Y -39.308,Z -81.339,A -90.000,B 90.000,C 0.000} C_DIS
LIN {X -24.384,Y -39.308,Z -81.098,A -90.000,B 90.000,C 0.000} C_DIS
LIN {X -22.800,Y -39.308,Z -79.364,A -90.000,B 90.000,C 0.000} C_DIS
LIN {X -22.308,Y -39.308,Z -78.836,A -90.000,B 90.000,C 0.000} C_DIS
LIN {X -20.794,Y -39.308,Z -77.477,A -90.000,B 90.000,C 0.000} C_DIS
LIN {X -20.549,Y -39.308,Z -77.271,A -90.000,B 90.000,C 0.000} C_DIS
LIN {X -20.138,Y -39.308,Z -76.949,A -90.000,B 90.000,C 0.000} C_DIS
LIN {X -19.639,Y -39.308,Z -76.600,A -90.000,B 90.000,C 0.000} C_DIS
LIN {X -19.365,Y -39.308,Z -76.435,A -90.000,B 90.000,C 0.000} C_DIS
LIN {X -18.624,Y -39.308,Z -76.033,A -90.000,B 90.000,C 0.000} C_DIS
LIN {X -18.017,Y -39.308,Z -75.755,A -90.000,B 90.000,C 0.000} C_DIS
LIN {X -17.429,Y -39.308,Z -75.519,A -90.000,B 90.000,C 0.000} C_DIS
LIN {X -16.976,Y -39.308,Z -75.350,A -90.000,B 90.000,C 0.000} C_DIS
LIN {X -16.706,Y -39.308,Z -75.269,A -90.000,B 90.000,C 0.000} C_DIS
LIN {X -15.733,Y -39.308,Z -74.988,A -90.000,B 90.000,C 0.000} C_DIS
LIN {X -15.601,Y -39.308,Z -74.950,A -90.000,B 90.000,C 0.000} C_DIS
LIN {X -15.290,Y -39.308,Z -74.878,A -90.000,B 90.000,C 0.000} C_DIS
LIN {X -14.940,Y -39.308,Z -74.830,A -90.000,B 90.000,C 0.000} C_DIS
LIN {X -14.714,Y -39.308,Z -74.809,A -90.000,B 90.000,C 0.000} C_DIS
LIN {X -14.395,Y -39.308,Z -74.786,A -90.000,B 90.000,C 0.000} C_DIS
LIN {X -12.689,Y -39.308,Z -74.741,A -90.000,B 90.000,C 0.000} C_DIS
LIN {X -11.256,Y -39.308,Z -74.743,A -90.000,B 90.000,C 0.000} C_DIS
LIN {X -10.422,Y -39.308,Z -74.795,A -90.000,B 90.000,C 0.000} C_DIS
LIN {X -8.342,Y -39.308,Z -74.961,A -90.000,B 90.000,C 0.000} C_DIS
LIN {X -8.253,Y -39.308,Z -74.969,A -90.000,B 90.000,C 0.000} C_DIS
LIN {X -7.377,Y -39.308,Z -75.068,A -90.000,B 90.000,C 0.000} C_DIS
LIN {X -4.616,Y -39.308,Z -75.581,A -90.000,B 90.000,C 0.000} C_DIS
LIN {X -3.025,Y -39.308,Z -75.860,A -90.000,B 90.000,C 0.000} C_DIS
LIN {X -1.814,Y -39.308,Z -76.126,A -90.000,B 90.000,C 0.000} C_DIS
LIN {X 0.586,Y -39.308,Z -76.628,A -90.000,B 90.000,C 0.000} C_DIS
LIN {X 1.164,Y -39.308,Z -76.755,A -90.000,B 90.000,C 0.000} C_DIS
LIN {X 1.413,Y -39.308,Z -76.805,A -90.000,B 90.000,C 0.000} C_DIS
LIN {X 3.924,Y -39.308,Z -77.408,A -90.000,B 90.000,C 0.000} C_DIS
LIN {X 5.837,Y -39.308,Z -77.827,A -90.000,B 90.000,C 0.000} C_DIS
LIN {X 6.788,Y -39.308,Z -78.065,A -90.000,B 90.000,C 0.000} C_DIS
LIN {X 7.699,Y -39.308,Z -78.286,A -90.000,B 90.000,C 0.000} C_DIS
LIN {X 8.954,Y -39.308,Z -78.541,A -90.000,B 90.000,C 0.000} C_DIS
LIN {X 10.021,Y -39.308,Z -78.721,A -90.000,B 90.000,C 0.000} C_DIS
LIN {X 10.647,Y -39.308,Z -78.860,A -90.000,B 90.000,C 0.000} C_DIS
LIN {X 10.802,Y -39.308,Z -78.893,A -90.000,B 90.000,C 0.000} C_DIS
LIN {X 11.687,Y -39.308,Z -78.893,A -90.000,B 90.000,C 0.000} C_DIS
LIN {X 12.238,Y -39.308,Z -78.860,A -90.000,B 90.000,C 0.000} C_DIS
LIN {X 12.581,Y -39.308,Z -78.689,A -90.000,B 90.000,C 0.000} C_DIS
LIN {X 13.037,Y -39.308,Z -78.435,A -90.000,B 90.000,C 0.000} C_DIS
LIN {X 13.252,Y -39.308,Z -78.154,A -90.000,B 90.000,C 0.000} C_DIS
LIN {X 13.769,Y -39.308,Z -77.553,A -90.000,B 90.000,C 0.000} C_DIS
LIN {X 14.076,Y -39.308,Z -77.229,A -90.000,B 90.000,C 0.000} C_DIS
LIN {X 14.202,Y -39.308,Z -77.101,A -90.000,B 90.000,C 0.000} C_DIS
LIN {X 14.935,Y -39.308,Z -76.630,A -90.000,B 90.000,C 0.000} C_DIS
LIN {X 15.091,Y -39.308,Z -76.542,A -90.000,B 90.000,C 0.000} C_DIS
LIN {X 15.266,Y -39.308,Z -76.499,A -90.000,B 90.000,C 0.000} C_DIS
LIN {X 15.751,Y -39.308,Z -76.394,A -90.000,B 90.000,C 0.000} C_DIS
LIN {X 15.988,Y -39.308,Z -76.391,A -90.000,B 90.000,C 0.000} C_DIS
LIN {X 16.419,Y -39.308,Z -76.422,A -90.000,B 90.000,C 0.000} C_DIS
LIN {X 18.031,Y -39.308,Z -76.509,A -90.000,B 90.000,C 0.000} C_DIS
LIN {X 17.965,Y -39.308,Z -76.441,A -90.000,B 90.000,C 0.000} C_DIS
LIN {X 17.672,Y -39.308,Z -76.047,A -90.000,B 90.000,C 0.000} C_DIS
LIN {X 17.575,Y -39.308,Z -75.907,A -90.000,B 90.000,C 0.000} C_DIS
LIN {X 16.850,Y -39.308,Z -74.742,A -90.000,B 90.000,C 0.000} C_DIS
LIN {X 16.576,Y -39.308,Z -74.221,A -90.000,B 90.000,C 0.000} C_DIS
LIN {X 16.428,Y -39.308,Z -73.817,A -90.000,B 90.000,C 0.000} C_DIS
LIN {X 16.297,Y -39.308,Z -73.229,A -90.000,B 90.000,C 0.000} C_DIS
LIN {X 16.149,Y -39.308,Z -72.541,A -90.000,B 90.000,C 0.000} C_DIS
LIN {X 16.050,Y -39.308,Z -71.857,A -90.000,B 90.000,C 0.000} C_DIS
LIN {X 16.029,Y -39.308,Z -71.506,A -90.000,B 90.000,C 0.000} C_DIS
LIN {X 16.035,Y -39.308,Z -71.341,A -90.000,B 90.000,C 0.000} C_DIS
LIN {X 16.065,Y -39.308,Z -71.002,A -90.000,B 90.000,C 0.000} C_DIS
LIN {X 16.115,Y -39.308,Z -70.781,A -90.000,B 90.000,C 0.000} C_DIS
LIN {X 16.143,Y -39.308,Z -70.671,A -90.000,B 90.000,C 0.000} C_DIS
LIN {X 16.225,Y -39.308,Z -70.460,A -90.000,B 90.000,C 0.000} C_DIS
LIN {X 16.269,Y -39.308,Z -70.355,A -90.000,B 90.000,C 0.000} C_DIS
LIN {X 16.366,Y -39.308,Z -70.166,A -90.000,B 90.000,C 0.000} C_DIS
LIN {X 16.535,Y -39.308,Z -69.896,A -90.000,B 90.000,C 0.000} C_DIS
LIN {X 16.745,Y -39.308,Z -69.655,A -90.000,B 90.000,C 0.000} C_DIS
LIN {X 16.990,Y -39.308,Z -69.450,A -90.000,B 90.000,C 0.000} C_DIS
LIN {X 17.264,Y -39.308,Z -69.285,A -90.000,B 90.000,C 0.000} C_DIS
LIN {X 17.560,Y -39.308,Z -69.165,A -90.000,B 90.000,C 0.000} C_DIS
LIN {X 17.673,Y -39.308,Z -69.138,A -90.000,B 90.000,C 0.000} C_DIS
LIN {X 18.130,Y -39.308,Z -68.974,A -90.000,B 90.000,C 0.000} C_DIS
LIN {X 18.441,Y -39.308,Z -68.902,A -90.000,B 90.000,C 0.000} C_DIS
LIN {X 18.503,Y -39.308,Z -68.889,A -90.000,B 90.000,C 0.000} C_DIS
LIN {X 18.831,Y -39.308,Z -68.867,A -90.000,B 90.000,C 0.000} C_DIS
LIN {X 19.210,Y -39.308,Z -68.893,A -90.000,B 90.000,C 0.000} C_DIS
LIN {X 19.463,Y -39.308,Z -68.913,A -90.000,B 90.000,C 0.000} C_DIS
LIN {X 19.806,Y -39.308,Z -68.990,A -90.000,B 90.000,C 0.000} C_DIS
LIN {X 20.270,Y -39.308,Z -69.113,A -90.000,B 90.000,C 0.000} C_DIS
LIN {X 20.830,Y -39.308,Z -69.297,A -90.000,B 90.000,C 0.000} C_DIS
LIN {X 21.121,Y -39.308,Z -69.400,A -90.000,B 90.000,C 0.000} C_DIS
LIN {X 21.568,Y -39.308,Z -69.577,A -90.000,B 90.000,C 0.000} C_DIS
LIN {X 21.578,Y -39.308,Z -69.468,A -90.000,B 90.000,C 0.000} C_DIS
LIN {X 21.600,Y -39.308,Z -69.352,A -90.000,B 90.000,C 0.000} C_DIS
LIN {X 21.665,Y -39.308,Z -69.050,A -90.000,B 90.000,C 0.000} C_DIS
LIN {X 21.687,Y -39.308,Z -68.965,A -90.000,B 90.000,C 0.000} C_DIS
LIN {X 21.800,Y -39.308,Z -68.695,A -90.000,B 90.000,C 0.000} C_DIS
LIN {X 21.957,Y -39.308,Z -68.449,A -90.000,B 90.000,C 0.000} C_DIS
LIN {X 22.041,Y -39.308,Z -68.331,A -90.000,B 90.000,C 0.000} C_DIS
LIN {X 22.127,Y -39.308,Z -68.233,A -90.000,B 90.000,C 0.000} C_DIS
LIN {X 22.240,Y -39.308,Z -68.111,A -90.000,B 90.000,C 0.000} C_DIS
LIN {X 22.340,Y -39.308,Z -68.027,A -90.000,B 90.000,C 0.000} C_DIS
LIN {X 22.474,Y -39.308,Z -67.927,A -90.000,B 90.000,C 0.000} C_DIS
LIN {X 22.585,Y -39.308,Z -67.860,A -90.000,B 90.000,C 0.000} C_DIS
LIN {X 22.735,Y -39.308,Z -67.785,A -90.000,B 90.000,C 0.000} C_DIS
LIN {X 22.855,Y -39.308,Z -67.736,A -90.000,B 90.000,C 0.000} C_DIS
LIN {X 23.081,Y -39.308,Z -67.670,A -90.000,B 90.000,C 0.000} C_DIS
LIN {X 23.393,Y -39.308,Z -67.598,A -90.000,B 90.000,C 0.000} C_DIS
LIN {X 23.711,Y -39.308,Z -67.575,A -90.000,B 90.000,C 0.000} C_DIS
LIN {X 24.223,Y -39.308,Z -67.589,A -90.000,B 90.000,C 0.000} C_DIS
LIN {X 24.574,Y -39.308,Z -67.617,A -90.000,B 90.000,C 0.000} C_DIS
LIN {X 24.611,Y -39.308,Z -67.622,A -90.000,B 90.000,C 0.000} C_DIS
LIN {X 24.836,Y -39.308,Z -67.668,A -90.000,B 90.000,C 0.000} C_DIS
LIN {X 25.085,Y -39.308,Z -67.723,A -90.000,B 90.000,C 0.000} C_DIS
LIN {X 25.701,Y -39.308,Z -67.890,A -90.000,B 90.000,C 0.000} C_DIS
LIN {X 25.806,Y -39.308,Z -67.921,A -90.000,B 90.000,C 0.000} C_DIS
LIN {X 26.166,Y -39.308,Z -68.039,A -90.000,B 90.000,C 0.000} C_DIS
LIN {X 26.589,Y -39.308,Z -68.197,A -90.000,B 90.000,C 0.000} C_DIS
LIN {X 26.834,Y -39.308,Z -68.301,A -90.000,B 90.000,C 0.000} C_DIS
LIN {X 26.963,Y -39.308,Z -68.153,A -90.000,B 90.000,C 0.000} C_DIS
LIN {X 27.095,Y -39.308,Z -68.013,A -90.000,B 90.000,C 0.000} C_DIS
LIN {X 27.357,Y -39.308,Z -67.781,A -90.000,B 90.000,C 0.000} C_DIS
LIN {X 27.849,Y -39.308,Z -67.417,A -90.000,B 90.000,C 0.000} C_DIS
LIN {X 28.154,Y -39.308,Z -67.229,A -90.000,B 90.000,C 0.000} C_DIS
LIN {X 28.500,Y -39.308,Z -67.056,A -90.000,B 90.000,C 0.000} C_DIS
LIN {X 28.542,Y -39.308,Z -67.037,A -90.000,B 90.000,C 0.000} C_DIS
LIN {X 28.483,Y -39.308,Z -65.705,A -90.000,B 90.000,C 0.000} C_DIS
LIN {X 28.472,Y -39.308,Z -65.475,A -90.000,B 90.000,C 0.000} C_DIS
LIN {X 28.445,Y -39.308,Z -64.382,A -90.000,B 90.000,C 0.000} C_DIS
LIN {X 28.437,Y -39.308,Z -63.685,A -90.000,B 90.000,C 0.000} C_DIS
LIN {X 28.447,Y -39.308,Z -63.244,A -90.000,B 90.000,C 0.000} C_DIS
LIN {X 28.471,Y -39.308,Z -62.551,A -90.000,B 90.000,C 0.000} C_DIS
LIN {X 28.498,Y -39.308,Z -62.202,A -90.000,B 90.000,C 0.000} C_DIS
LIN {X 28.553,Y -39.308,Z -61.782,A -90.000,B 90.000,C 0.000} C_DIS
LIN {X 28.616,Y -39.308,Z -61.373,A -90.000,B 90.000,C 0.000} C_DIS
LIN {X 28.662,Y -39.308,Z -61.082,A -90.000,B 90.000,C 0.000} C_DIS
LIN {X 28.692,Y -39.308,Z -60.902,A -90.000,B 90.000,C 0.000} C_DIS
LIN {X 28.703,Y -39.308,Z -60.848,A -90.000,B 90.000,C 0.000} C_DIS
LIN {X 28.782,Y -39.308,Z -60.504,A -90.000,B 90.000,C 0.000} C_DIS
LIN {X 28.809,Y -39.308,Z -60.397,A -90.000,B 90.000,C 0.000} C_DIS
LIN {X 28.947,Y -39.308,Z -60.019,A -90.000,B 90.000,C 0.000} C_DIS
LIN {X 29.073,Y -39.308,Z -59.729,A -90.000,B 90.000,C 0.000} C_DIS
LIN {X 29.234,Y -39.308,Z -59.386,A -90.000,B 90.000,C 0.000} C_DIS
LIN {X 29.439,Y -39.308,Z -59.067,A -90.000,B 90.000,C 0.000} C_DIS
LIN {X 29.750,Y -39.308,Z -58.661,A -90.000,B 90.000,C 0.000} C_DIS
LIN {X 30.001,Y -39.308,Z -58.415,A -90.000,B 90.000,C 0.000} C_DIS
LIN {X 30.306,Y -39.308,Z -58.190,A -90.000,B 90.000,C 0.000} C_DIS
LIN {X 30.484,Y -39.308,Z -58.070,A -90.000,B 90.000,C 0.000} C_DIS
LIN {X 30.794,Y -39.308,Z -57.905,A -90.000,B 90.000,C 0.000} C_DIS
LIN {X 31.124,Y -39.308,Z -57.784,A -90.000,B 90.000,C 0.000} C_DIS
LIN {X 31.496,Y -39.308,Z -57.707,A -90.000,B 90.000,C 0.000} C_DIS
LIN {X 31.799,Y -39.308,Z -57.670,A -90.000,B 90.000,C 0.000} C_DIS
LIN {X 31.962,Y -39.308,Z -57.659,A -90.000,B 90.000,C 0.000} C_DIS
LIN {X 32.074,Y -39.308,Z -57.186,A -90.000,B 90.000,C 0.000} C_DIS
LIN {X 32.278,Y -39.308,Z -56.528,A -90.000,B 90.000,C 0.000} C_DIS
LIN {X 32.331,Y -39.308,Z -56.329,A -90.000,B 90.000,C 0.000} C_DIS
LIN {X 32.489,Y -39.308,Z -55.802,A -90.000,B 90.000,C 0.000} C_DIS
LIN {X 32.645,Y -39.308,Z -55.390,A -90.000,B 90.000,C 0.000} C_DIS
LIN {X 32.823,Y -39.308,Z -55.001,A -90.000,B 90.000,C 0.000} C_DIS
LIN {X 32.854,Y -39.308,Z -54.941,A -90.000,B 90.000,C 0.000} C_DIS
LIN {X 32.910,Y -39.308,Z -54.828,A -90.000,B 90.000,C 0.000} C_DIS
LIN {X 33.112,Y -39.308,Z -54.443,A -90.000,B 90.000,C 0.000} C_DIS
LIN {X 33.165,Y -39.308,Z -54.325,A -90.000,B 90.000,C 0.000} C_DIS
LIN {X 33.362,Y -39.308,Z -53.951,A -90.000,B 90.000,C 0.000} C_DIS
LIN {X 33.603,Y -39.308,Z -53.602,A -90.000,B 90.000,C 0.000} C_DIS
LIN {X 33.932,Y -39.308,Z -53.214,A -90.000,B 90.000,C 0.000} C_DIS
LIN {X 34.127,Y -39.308,Z -52.952,A -90.000,B 90.000,C 0.000} C_DIS
LIN {X 34.180,Y -39.308,Z -52.882,A -90.000,B 90.000,C 0.000} C_DIS
LIN {X 34.447,Y -39.308,Z -52.580,A -90.000,B 90.000,C 0.000} C_DIS
LIN {X 34.749,Y -39.308,Z -52.313,A -90.000,B 90.000,C 0.000} C_DIS
LIN {X 34.968,Y -39.308,Z -52.140,A -90.000,B 90.000,C 0.000} C_DIS
LIN {X 35.338,Y -39.308,Z -51.820,A -90.000,B 90.000,C 0.000} C_DIS
LIN {X 35.671,Y -39.308,Z -51.592,A -90.000,B 90.000,C 0.000} C_DIS
LIN {X 36.029,Y -39.308,Z -51.407,A -90.000,B 90.000,C 0.000} C_DIS
LIN {X 36.235,Y -39.308,Z -51.312,A -90.000,B 90.000,C 0.000} C_DIS
LIN {X 36.760,Y -39.308,Z -51.057,A -90.000,B 90.000,C 0.000} C_DIS
LIN {X 37.138,Y -39.308,Z -50.918,A -90.000,B 90.000,C 0.000} C_DIS
LIN {X 37.531,Y -39.308,Z -50.827,A -90.000,B 90.000,C 0.000} C_DIS
LIN {X 38.416,Y -39.308,Z -50.672,A -90.000,B 90.000,C 0.000} C_DIS
LIN {X 38.817,Y -39.308,Z -50.630,A -90.000,B 90.000,C 0.000} C_DIS
LIN {X 39.220,Y -39.308,Z -50.638,A -90.000,B 90.000,C 0.000} C_DIS
LIN {X 40.269,Y -39.308,Z -50.731,A -90.000,B 90.000,C 0.000} C_DIS
LIN {X 40.736,Y -39.308,Z -50.783,A -90.000,B 90.000,C 0.000} C_DIS
LIN {X 41.150,Y -39.308,Z -50.873,A -90.000,B 90.000,C 0.000} C_DIS
LIN {X 41.568,Y -39.308,Z -51.007,A -90.000,B 90.000,C 0.000} C_DIS
LIN {X 42.363,Y -39.308,Z -51.270,A -90.000,B 90.000,C 0.000} C_DIS
LIN {X 42.831,Y -39.308,Z -51.432,A -90.000,B 90.000,C 0.000} C_DIS
LIN {X 43.231,Y -39.308,Z -51.591,A -90.000,B 90.000,C 0.000} C_DIS
LIN {X 43.883,Y -39.308,Z -51.857,A -90.000,B 90.000,C 0.000} C_DIS
LIN {X 44.108,Y -39.308,Z -51.966,A -90.000,B 90.000,C 0.000} C_DIS
LIN {X 44.934,Y -39.308,Z -52.324,A -90.000,B 90.000,C 0.000} C_DIS
LIN {X 45.042,Y -39.308,Z -52.373,A -90.000,B 90.000,C 0.000} C_DIS
LIN {X 45.477,Y -39.308,Z -52.489,A -90.000,B 90.000,C 0.000} C_DIS
LIN {X 46.199,Y -39.308,Z -52.447,A -90.000,B 90.000,C 0.000} C_DIS
LIN {X 46.410,Y -39.308,Z -52.419,A -90.000,B 90.000,C 0.000} C_DIS
LIN {X 47.570,Y -39.308,Z -52.251,A -90.000,B 90.000,C 0.000} C_DIS
LIN {X 47.948,Y -39.308,Z -52.222,A -90.000,B 90.000,C 0.000} C_DIS
LIN {X 48.294,Y -39.308,Z -52.223,A -90.000,B 90.000,C 0.000} C_DIS
LIN {X 49.620,Y -39.308,Z -52.195,A -90.000,B 90.000,C 0.000} C_DIS
LIN {X 49.998,Y -39.308,Z -52.216,A -90.000,B 90.000,C 0.000} C_DIS
LIN {X 50.371,Y -39.308,Z -52.286,A -90.000,B 90.000,C 0.000} C_DIS
LIN {X 50.891,Y -39.308,Z -52.444,A -90.000,B 90.000,C 0.000} C_DIS
LIN {X 52.245,Y -39.308,Z -52.814,A -90.000,B 90.000,C 0.000} C_DIS
LIN {X 52.605,Y -39.308,Z -52.933,A -90.000,B 90.000,C 0.000} C_DIS
LIN {X 52.946,Y -39.308,Z -53.098,A -90.000,B 90.000,C 0.000} C_DIS
LIN {X 53.320,Y -39.308,Z -53.319,A -90.000,B 90.000,C 0.000} C_DIS
LIN {X 54.566,Y -39.308,Z -54.219,A -90.000,B 90.000,C 0.000} C_DIS
LIN {X 55.348,Y -39.308,Z -54.749,A -90.000,B 90.000,C 0.000} C_DIS
LIN {X 55.671,Y -39.308,Z -54.990,A -90.000,B 90.000,C 0.000} C_DIS
LIN {X 55.961,Y -39.308,Z -55.269,A -90.000,B 90.000,C 0.000} C_DIS
LIN {X 57.932,Y -39.308,Z -57.235,A -90.000,B 90.000,C 0.000} C_DIS
LIN {X 58.007,Y -39.308,Z -57.308,A -90.000,B 90.000,C 0.000} C_DIS
LIN {X 58.083,Y -39.308,Z -57.399,A -90.000,B 90.000,C 0.000} C_DIS
LIN {X 58.338,Y -39.308,Z -57.712,A -90.000,B 90.000,C 0.000} C_DIS
LIN {X 58.939,Y -39.308,Z -58.498,A -90.000,B 90.000,C 0.000} C_DIS
LIN {X 59.973,Y -39.308,Z -60.001,A -90.000,B 90.000,C 0.000} C_DIS
LIN {X 60.112,Y -39.308,Z -60.207,A -90.000,B 90.000,C 0.000} C_DIS
LIN {X 61.437,Y -39.308,Z -62.377,A -90.000,B 90.000,C 0.000} C_DIS
LIN {X 61.766,Y -39.308,Z -63.019,A -90.000,B 90.000,C 0.000} C_DIS
LIN {X 62.295,Y -39.308,Z -64.004,A -90.000,B 90.000,C 0.000} C_DIS
LIN {X 63.304,Y -39.308,Z -65.901,A -90.000,B 90.000,C 0.000} C_DIS
LIN {X 63.329,Y -39.308,Z -65.960,A -90.000,B 90.000,C 0.000} C_DIS
LIN {X 63.952,Y -39.308,Z -67.049,A -90.000,B 90.000,C 0.000} C_DIS
LIN {X 64.697,Y -39.308,Z -68.012,A -90.000,B 90.000,C 0.000} C_DIS
LIN {X 64.899,Y -39.308,Z -68.283,A -90.000,B 90.000,C 0.000} C_DIS
LIN {X 64.951,Y -39.308,Z -68.361,A -90.000,B 90.000,C 0.000} C_DIS
LIN {X 65.300,Y -39.308,Z -68.822,A -90.000,B 90.000,C 0.000} C_DIS
LIN {X 65.685,Y -39.308,Z -69.338,A -90.000,B 90.000,C 0.000} C_DIS
LIN {X 66.429,Y -39.308,Z -70.040,A -90.000,B 90.000,C 0.000} C_DIS
LIN {X 66.666,Y -39.308,Z -70.279,A -90.000,B 90.000,C 0.000} C_DIS
LIN {X 66.766,Y -39.308,Z -70.390,A -90.000,B 90.000,C 0.000} C_DIS
LIN {X 67.264,Y -39.308,Z -70.816,A -90.000,B 90.000,C 0.000} C_DIS
LIN {X 68.013,Y -39.308,Z -71.562,A -90.000,B 90.000,C 0.000} C_DIS
LIN {X 68.267,Y -39.308,Z -71.753,A -90.000,B 90.000,C 0.000} C_DIS
LIN {X 69.278,Y -39.308,Z -72.580,A -90.000,B 90.000,C 0.000} C_DIS
LIN {X 69.974,Y -39.308,Z -73.200,A -90.000,B 90.000,C 0.000} C_DIS
LIN {X 70.414,Y -39.308,Z -73.564,A -90.000,B 90.000,C 0.000} C_DIS
LIN {X 71.621,Y -39.308,Z -74.574,A -90.000,B 90.000,C 0.000} C_DIS
LIN {X 72.481,Y -39.308,Z -75.351,A -90.000,B 90.000,C 0.000} C_DIS
LIN {X 72.729,Y -39.308,Z -75.600,A -90.000,B 90.000,C 0.000} C_DIS
LIN {X 72.880,Y -39.308,Z -75.759,A -90.000,B 90.000,C 0.000} C_DIS
LIN {X 73.139,Y -39.308,Z -75.972,A -90.000,B 90.000,C 0.000} C_DIS
LIN {X 73.587,Y -39.308,Z -76.406,A -90.000,B 90.000,C 0.000} C_DIS
LIN {X 73.725,Y -39.308,Z -76.560,A -90.000,B 90.000,C 0.000} C_DIS
LIN {X 73.866,Y -39.308,Z -76.691,A -90.000,B 90.000,C 0.000} C_DIS
LIN {X 74.285,Y -39.308,Z -77.141,A -90.000,B 90.000,C 0.000} C_DIS
LIN {X 74.383,Y -39.308,Z -77.250,A -90.000,B 90.000,C 0.000} C_DIS
LIN {X 74.503,Y -39.308,Z -77.352,A -90.000,B 90.000,C 0.000} C_DIS
LIN {X 74.977,Y -39.308,Z -77.790,A -90.000,B 90.000,C 0.000} C_DIS
LIN {X 75.106,Y -39.308,Z -77.932,A -90.000,B 90.000,C 0.000} C_DIS
LIN {X 75.293,Y -39.308,Z -78.094,A -90.000,B 90.000,C 0.000} C_DIS
LIN {X 75.577,Y -39.308,Z -78.378,A -90.000,B 90.000,C 0.000} C_DIS
LIN {X 75.901,Y -39.308,Z -78.612,A -90.000,B 90.000,C 0.000} C_DIS
LIN {X 76.067,Y -39.308,Z -78.755,A -90.000,B 90.000,C 0.000} C_DIS
LIN {X 76.118,Y -39.308,Z -78.785,A -90.000,B 90.000,C 0.000} C_DIS
LIN {X 76.441,Y -39.308,Z -78.997,A -90.000,B 90.000,C 0.000} C_DIS
LIN {X 76.656,Y -39.308,Z -79.102,A -90.000,B 90.000,C 0.000} C_DIS
LIN {X 76.688,Y -39.308,Z -79.120,A -90.000,B 90.000,C 0.000} C_DIS
LIN {X 76.710,Y -39.308,Z -79.125,A -90.000,B 90.000,C 0.000} C_DIS
LIN {X 77.161,Y -39.308,Z -79.167,A -90.000,B 90.000,C 0.000} C_DIS
LIN {X 77.559,Y -39.308,Z -79.090,A -90.000,B 90.000,C 0.000} C_DIS
LIN {X 77.612,Y -39.308,Z -79.084,A -90.000,B 90.000,C 0.000} C_DIS
LIN {X 77.977,Y -39.308,Z -79.016,A -90.000,B 90.000,C 0.000} C_DIS
LIN {X 78.290,Y -39.308,Z -78.938,A -90.000,B 90.000,C 0.000} C_DIS
LIN {X 78.412,Y -39.308,Z -78.912,A -90.000,B 90.000,C 0.000} C_DIS
LIN {X 78.545,Y -39.308,Z -78.873,A -90.000,B 90.000,C 0.000} C_DIS
LIN {X 78.835,Y -39.308,Z -78.806,A -90.000,B 90.000,C 0.000} C_DIS
LIN {X 78.849,Y -39.308,Z -78.800,A -90.000,B 90.000,C 0.000} C_DIS
LIN {X 78.919,Y -39.308,Z -78.422,A -90.000,B 90.000,C 0.000} C_DIS
LIN {X 78.918,Y -39.308,Z -78.145,A -90.000,B 90.000,C 0.000} C_DIS
LIN {X 78.928,Y -39.308,Z -77.704,A -90.000,B 90.000,C 0.000} C_DIS
LIN {X 78.966,Y -39.308,Z -77.105,A -90.000,B 90.000,C 0.000} C_DIS
LIN {X 78.949,Y -39.308,Z -76.200,A -90.000,B 90.000,C 0.000} C_DIS
LIN {X 78.896,Y -39.308,Z -75.357,A -90.000,B 90.000,C 0.000} C_DIS
LIN {X 78.895,Y -39.308,Z -74.983,A -90.000,B 90.000,C 0.000} C_DIS
LIN {X 78.880,Y -39.308,Z -74.674,A -90.000,B 90.000,C 0.000} C_DIS
LIN {X 78.841,Y -39.308,Z -72.479,A -90.000,B 90.000,C 0.000} C_DIS
LIN {X 78.851,Y -39.308,Z -71.941,A -90.000,B 90.000,C 0.000} C_DIS
LIN {X 78.873,Y -39.308,Z -71.465,A -90.000,B 90.000,C 0.000} C_DIS
LIN {X 78.963,Y -39.308,Z -70.545,A -90.000,B 90.000,C 0.000} C_DIS
LIN {X 78.980,Y -39.308,Z -70.392,A -90.000,B 90.000,C 0.000} C_DIS
LIN {X 79.071,Y -39.308,Z -69.918,A -90.000,B 90.000,C 0.000} C_DIS
LIN {X 79.117,Y -39.308,Z -69.703,A -90.000,B 90.000,C 0.000} C_DIS
LIN {X 79.245,Y -39.308,Z -69.069,A -90.000,B 90.000,C 0.000} C_DIS
LIN {X 79.340,Y -39.308,Z -68.644,A -90.000,B 90.000,C 0.000} C_DIS
LIN {X 79.688,Y -39.308,Z -67.582,A -90.000,B 90.000,C 0.000} C_DIS
LIN {X 79.789,Y -39.308,Z -67.300,A -90.000,B 90.000,C 0.000} C_DIS
LIN {X 79.866,Y -39.308,Z -67.094,A -90.000,B 90.000,C 0.000} C_DIS
LIN {X 79.920,Y -39.308,Z -66.965,A -90.000,B 90.000,C 0.000} C_DIS
LIN {X 80.458,Y -39.308,Z -65.744,A -90.000,B 90.000,C 0.000} C_DIS
LIN {X 80.645,Y -39.308,Z -65.334,A -90.000,B 90.000,C 0.000} C_DIS
LIN {X 81.438,Y -39.308,Z -63.804,A -90.000,B 90.000,C 0.000} C_DIS
LIN {X 81.709,Y -39.308,Z -63.342,A -90.000,B 90.000,C 0.000} C_DIS
LIN {X 82.705,Y -39.308,Z -61.742,A -90.000,B 90.000,C 0.000} C_DIS
LIN {X 84.243,Y -39.308,Z -59.630,A -90.000,B 90.000,C 0.000} C_DIS
LIN {X 85.732,Y -39.308,Z -57.856,A -90.000,B 90.000,C 0.000} C_DIS
LIN {X 86.059,Y -39.308,Z -57.494,A -90.000,B 90.000,C 0.000} C_DIS
LIN {X 87.795,Y -39.308,Z -55.685,A -90.000,B 90.000,C 0.000} C_DIS
LIN {X 89.945,Y -39.308,Z -53.719,A -90.000,B 90.000,C 0.000} C_DIS
LIN {X 90.159,Y -39.308,Z -53.526,A -90.000,B 90.000,C 0.000} C_DIS
LIN {X 92.365,Y -39.308,Z -51.637,A -90.000,B 90.000,C 0.000} C_DIS
LIN {X 94.367,Y -39.308,Z -49.945,A -90.000,B 90.000,C 0.000} C_DIS
LIN {X 96.070,Y -39.308,Z -48.453,A -90.000,B 90.000,C 0.000} C_DIS
LIN {X 96.910,Y -39.308,Z -47.638,A -90.000,B 90.000,C 0.000} C_DIS
LIN {X 97.648,Y -39.308,Z -46.921,A -90.000,B 90.000,C 0.000} C_DIS
LIN {X 99.081,Y -39.308,Z -45.409,A -90.000,B 90.000,C 0.000} C_DIS
LIN {X 100.086,Y -39.308,Z -44.290,A -90.000,B 90.000,C 0.000} C_DIS
LIN {X 101.207,Y -39.308,Z -43.025,A -90.000,B 90.000,C 0.000} C_DIS
